LIN {X 0,Y 281.063,Z 426.792,A -85,B 0,C 180,E1 12589.746,E2 12589.746} C_VEL
LIN {X 0,Y 283.096,Z 428.214,A -85,B 0,C 180,E1 12587.55,E2 12587.55} C_VEL
LIN {X 0,Y 285.507,Z 432.072,A -85,B 0,C 180,E1 12585.18,E2 12585.18} C_VEL
LIN {X 0,Y 287.987,Z 434.4,A -85,B 0,C 180,E1 12583.244,E2 12583.244} C_VEL
LIN {X 0,Y 291.212,Z 438.721,A -85,B 0,C 180,E1 12580.955,E2 12580.955} C_VEL
LIN {X 0,Y 292.622,Z 440.371,A -85,B 0,C 180,E1 12580.065,E2 12580.065} C_VEL
LIN {X 0,Y 296.342,Z 445.028,A -85,B 0,C 180,E1 12577.894,E2 12577.894} C_VEL
LIN {X 0,Y 301.456,Z 452.142,A -85,B 0,C 180,E1 12575.238,E2 12575.238} C_VEL
LIN {X 0,Y 306.819,Z 459.539,A -85,B 0,C 180,E1 12572.796,E2 12572.796} C_VEL
LIN {X 0,Y 313.495,Z 471.371,A -85,B 0,C 180,E1 12569.997,E2 12569.997} C_VEL
LIN {X 0,Y 320.303,Z 484.326,A -85,B 0,C 180,E1 12567.438,E2 12567.438} C_VEL
LIN {X 0,Y 324.467,Z 493.018,A -85,B 0,C 180,E1 12565.976,E2 12565.976} C_VEL
LIN {X 0,Y 324.937,Z 495.745,A -85,B 0,C 180,E1 12565.75,E2 12565.75} C_VEL
LIN {X 0,Y 324.322,Z 500.372,A -85,B 0,C 180,E1 12565.731,E2 12565.731} C_VEL
LIN {X 0,Y 320.258,Z 513.224,A -85,B 0,C 180,E1 12566.295,E2 12566.295} C_VEL
LIN {X 0,Y 319.782,Z 516.489,A -85,B 0,C 180,E1 12566.293,E2 12566.293} C_VEL
LIN {X 0,Y 311.091,Z 643.63,A -85,B 0,C 180,E1 12563.53,E2 12563.53} C_VEL
LIN {X 0,Y 308.318,Z 665.175,A -85,B 0,C 180,E1 12562.857,E2 12562.857} C_VEL
LIN {X 0,Y 304.957,Z 682.984,A -85,B 0,C 180,E1 12562.072,E2 12562.072} C_VEL
LIN {X 0,Y 301.16,Z 699.447,A -85,B 0,C 180,E1 12561.128,E2 12561.128} C_VEL
LIN {X 0,Y 296.032,Z 718.293,A -85,B 0,C 180,E1 12559.756,E2 12559.756} C_VEL
LIN {X 0,Y 290.238,Z 736.04,A -85,B 0,C 180,E1 12558.081,E2 12558.081} C_VEL
LIN {X 0,Y 285.027,Z 750.363,A -85,B 0,C 180,E1 12556.437,E2 12556.437} C_VEL
LIN {X 0,Y 278.742,Z 766.216,A -85,B 0,C 180,E1 12554.239,E2 12554.239} C_VEL
LIN {X 0,Y 271.755,Z 782.159,A -85,B 0,C 180,E1 12551.472,E2 12551.472} C_VEL
LIN {X 0,Y 266.062,Z 794.478,A -85,B 0,C 180,E1 12548.871,E2 12548.871} C_VEL
LIN {X 0,Y 259.825,Z 807.626,A -85,B 0,C 180,E1 12545.525,E2 12545.525} C_VEL
LIN {X 0,Y 254.077,Z 819.333,A -85,B 0,C 180,E1 12541.775,E2 12541.775} C_VEL
LIN {X 0,Y 249.789,Z 828.338,A -85,B 0,C 180,E1 12538.27,E2 12538.27} C_VEL
LIN {X 0,Y 245.803,Z 837.325,A -85,B 0,C 180,E1 12534.002,E2 12534.002} C_VEL
LIN {X 0,Y 242.846,Z 844.673,A -85,B 0,C 180,E1 12529.445,E2 12529.445} C_VEL
LIN {X 0,Y 241.192,Z 849.808,A -85,B 0,C 180,E1 12525.385,E2 12525.385} C_VEL
LIN {X 0,Y 240.239,Z 854.173,A -85,B 0,C 180,E1 12520.788,E2 12520.788} C_VEL
LIN {X 0,Y 239.969,Z 856.979,A -85,B 0,C 180,E1 12515.979,E2 12515.979} C_VEL
LIN {X 0,Y 239.985,Z 858.077,A -85,B 0,C 180,E1 12512.149,E2 12512.149} C_VEL
LIN {X 0,Y 239.995,Z 858.167,A -85,B 0,C 180,E1 12508.568,E2 12508.568} C_VEL
LIN {X 0,Y 239.966,Z 857.285,A -85,B 0,C 180,E1 12504.836,E2 12504.836} C_VEL
LIN {X 0,Y 240.065,Z 855.439,A -85,B 0,C 180,E1 12501.136,E2 12501.136} C_VEL
LIN {X 0,Y 240.583,Z 852.272,A -85,B 0,C 180,E1 12497.031,E2 12497.031} C_VEL
LIN {X 0,Y 242.18,Z 846.644,A -85,B 0,C 180,E1 12491.963,E2 12491.963} C_VEL
LIN {X 0,Y 244.58,Z 840.152,A -85,B 0,C 180,E1 12487.655,E2 12487.655} C_VEL
LIN {X 0,Y 247.831,Z 832.624,A -85,B 0,C 180,E1 12483.655,E2 12483.655} C_VEL
LIN {X 0,Y 252.943,Z 821.703,A -85,B 0,C 180,E1 12479.079,E2 12479.079} C_VEL
LIN {X 0,Y 257.756,Z 811.744,A -85,B 0,C 180,E1 12475.726,E2 12475.726} C_VEL
LIN {X 0,Y 263.28,Z 800.376,A -85,B 0,C 180,E1 12472.545,E2 12472.545} C_VEL
LIN {X 0,Y 270.176,Z 785.665,A -85,B 0,C 180,E1 12469.219,E2 12469.219} C_VEL
LIN {X 0,Y 276.002,Z 772.517,A -85,B 0,C 180,E1 12466.791,E2 12466.791} C_VEL
LIN {X 0,Y 282.337,Z 757.376,A -85,B 0,C 180,E1 12464.474,E2 12464.474} C_VEL
LIN {X 0,Y 288.83,Z 740.076,A -85,B 0,C 180,E1 12462.348,E2 12462.348} C_VEL
LIN {X 0,Y 293.964,Z 724.757,A -85,B 0,C 180,E1 12460.82,E2 12460.82} C_VEL
LIN {X 0,Y 298.845,Z 708.319,A -85,B 0,C 180,E1 12459.479,E2 12459.479} C_VEL
LIN {X 0,Y 303.971,Z 687.7,A -85,B 0,C 180,E1 12458.175,E2 12458.175} C_VEL
LIN {X 0,Y 307.421,Z 670.269,A -85,B 0,C 180,E1 12457.351,E2 12457.351} C_VEL
LIN {X 0,Y 310.141,Z 652.377,A -85,B 0,C 180,E1 12456.715,E2 12456.715} C_VEL
LIN {X 0,Y 312.495,Z 625.497,A -85,B 0,C 180,E1 12456.047,E2 12456.047} C_VEL
LIN {X 0,Y 320.903,Z 498.988,A -85,B 0,C 180,E1 12453.315,E2 12453.315} C_VEL
LIN {X 0,Y 314.641,Z 485.874,A -85,B 0,C 180,E1 12450.991,E2 12450.991} C_VEL
LIN {X 0,Y 307.924,Z 473.075,A -85,B 0,C 180,E1 12448.253,E2 12448.253} C_VEL
LIN {X 0,Y 303.272,Z 465.071,A -85,B 0,C 180,E1 12446.172,E2 12446.172} C_VEL
LIN {X 0,Y 297.362,Z 456.629,A -85,B 0,C 180,E1 12443.279,E2 12443.279} C_VEL
LIN {X 0,Y 293.549,Z 451.571,A -85,B 0,C 180,E1 12441.172,E2 12441.172} C_VEL
LIN {X 0,Y 289.811,Z 446.551,A -85,B 0,C 180,E1 12438.827,E2 12438.827} C_VEL
LIN {X 0,Y 286.373,Z 441.99,A -85,B 0,C 180,E1 12436.331,E2 12436.331} C_VEL
LIN {X 0,Y 282.436,Z 437.446,A -85,B 0,C 180,E1 12432.895,E2 12432.895} C_VEL
LIN {X 0,Y 281.366,Z 435.538,A -85,B 0,C 180,E1 12431.695,E2 12431.695} C_VEL
LIN {X 0,Y 278.26,Z 432.838,A -85,B 0,C 180,E1 12427.649,E2 12427.649} C_VEL
LIN {X 0,Y 276.894,Z 429.844,A -85,B 0,C 180,E1 12424.358,E2 12424.358} C_VEL
LIN {X 0,Y 276.092,Z 429.238,A -85,B 0,C 180,E1 12420.009,E2 12420.009} C_VEL
LIN {X 0,Y 276.821,Z 429.756,A -85,B 0,C 180,E1 12415.452,E2 12415.452} C_VEL
LIN {X 0,Y 280.254,Z 434.876,A -85,B 0,C 180,E1 12409.11,E2 12409.11} C_VEL
LIN {X 0,Y 281.805,Z 436.112,A -85,B 0,C 180,E1 12407.406,E2 12407.406} C_VEL
LIN {X 0,Y 284.403,Z 440.099,A -85,B 0,C 180,E1 12404.826,E2 12404.826} C_VEL
LIN {X 0,Y 286.349,Z 442.006,A -85,B 0,C 180,E1 12403.268,E2 12403.268} C_VEL
LIN {X 0,Y 289.491,Z 446.297,A -85,B 0,C 180,E1 12400.961,E2 12400.961} C_VEL
LIN {X 0,Y 290.943,Z 448.031,A -85,B 0,C 180,E1 12400.015,E2 12400.015} C_VEL
LIN {X 0,Y 295.057,Z 453.594,A -85,B 0,C 180,E1 12397.549,E2 12397.549} C_VEL
LIN {X 0,Y 301.079,Z 461.013,A -85,B 0,C 180,E1 12394.487,E2 12394.487} C_VEL
LIN {X 0,Y 306.421,Z 466.113,A -85,B 0,C 180,E1 12392.197,E2 12392.197} C_VEL
LIN {X 0,Y 312.519,Z 471.944,A -85,B 0,C 180,E1 12389.647,E2 12389.647} C_VEL
LIN {X 0,Y 317.174,Z 475.591,A -85,B 0,C 180,E1 12387.606,E2 12387.606} C_VEL
LIN {X 0,Y 322.098,Z 480.221,A -85,B 0,C 180,E1 12385.18,E2 12385.18} C_VEL
LIN {X 0,Y 325.293,Z 482.787,A -85,B 0,C 180,E1 12383.517,E2 12383.517} C_VEL
LIN {X 0,Y 329.435,Z 487.109,A -85,B 0,C 180,E1 12381.091,E2 12381.091} C_VEL
LIN {X 0,Y 332.913,Z 490.098,A -85,B 0,C 180,E1 12379,E2 12379} C_VEL
LIN {X 0,Y 337.324,Z 494.746,A -85,B 0,C 180,E1 12376.216,E2 12376.216} C_VEL
LIN {X 0,Y 340.322,Z 497.124,A -85,B 0,C 180,E1 12374.339,E2 12374.339} C_VEL
LIN {X 0,Y 344.324,Z 501.472,A -85,B 0,C 180,E1 12371.633,E2 12371.633} C_VEL
LIN {X 0,Y 348.17,Z 504.479,A -85,B 0,C 180,E1 12369.047,E2 12369.047} C_VEL
LIN {X 0,Y 352.251,Z 508.897,A -85,B 0,C 180,E1 12366.023,E2 12366.023} C_VEL
LIN {X 0,Y 356.277,Z 511.889,A -85,B 0,C 180,E1 12362.972,E2 12362.972} C_VEL
LIN {X 0,Y 359.522,Z 515.605,A -85,B 0,C 180,E1 12360.223,E2 12360.223} C_VEL
LIN {X 0,Y 362.97,Z 518.189,A -85,B 0,C 180,E1 12357.21,E2 12357.21} C_VEL
LIN {X 0,Y 364.703,Z 519.278,A -85,B 0,C 180,E1 12355.606,E2 12355.606} C_VEL
LIN {X 0,Y 367.351,Z 522.689,A -85,B 0,C 180,E1 12352.705,E2 12352.705} C_VEL
LIN {X 0,Y 370.191,Z 525.054,A -85,B 0,C 180,E1 12349.403,E2 12349.403} C_VEL
LIN {X 0,Y 372.765,Z 526.313,A -85,B 0,C 180,E1 12346.037,E2 12346.037} C_VEL
LIN {X 0,Y 373.961,Z 527.419,A -85,B 0,C 180,E1 12344.081,E2 12344.081} C_VEL
LIN {X 0,Y 375.427,Z 529.663,A -85,B 0,C 180,E1 12341.055,E2 12341.055} C_VEL
LIN {X 0,Y 376.685,Z 531.057,A -85,B 0,C 180,E1 12337.78,E2 12337.78} C_VEL
LIN {X 0,Y 377.57,Z 531.82,A -85,B 0,C 180,E1 12334.404,E2 12334.404} C_VEL
LIN {X 0,Y 377.93,Z 532.086,A -85,B 0,C 180,E1 12330.975,E2 12330.975} C_VEL
LIN {X 0,Y 377.84,Z 532.043,A -85,B 0,C 180,E1 12327.573,E2 12327.573} C_VEL
LIN {X 0,Y 377.25,Z 531.557,A -85,B 0,C 180,E1 12324.22,E2 12324.22} C_VEL
LIN {X 0,Y 376.186,Z 530.598,A -85,B 0,C 180,E1 12320.824,E2 12320.824} C_VEL
LIN {X 0,Y 374.776,Z 528.735,A -85,B 0,C 180,E1 12317.49,E2 12317.49} C_VEL
LIN {X 0,Y 373.168,Z 526.505,A -85,B 0,C 180,E1 12314.618,E2 12314.618} C_VEL
LIN {X 0,Y 370.673,Z 525.343,A -85,B 0,C 180,E1 12311.192,E2 12311.192} C_VEL
LIN {X 0,Y 367.915,Z 523.228,A -85,B 0,C 180,E1 12307.9,E2 12307.9} C_VEL
LIN {X 0,Y 365.196,Z 520.086,A -85,B 0,C 180,E1 12304.965,E2 12304.965} C_VEL
LIN {X 0,Y 364.121,Z 518.785,A -85,B 0,C 180,E1 12303.863,E2 12303.863} C_VEL
LIN {X 0,Y 360.72,Z 516.653,A -85,B 0,C 180,E1 12300.802,E2 12300.802} C_VEL
LIN {X 0,Y 357.303,Z 513.23,A -85,B 0,C 180,E1 12297.882,E2 12297.882} C_VEL
LIN {X 0,Y 355.438,Z 511.103,A -85,B 0,C 180,E1 12296.354,E2 12296.354} C_VEL
LIN {X 0,Y 351.656,Z 508.36,A -85,B 0,C 180,E1 12293.542,E2 12293.542} C_VEL
LIN {X 0,Y 347.13,Z 503.534,A -85,B 0,C 180,E1 12290.251,E2 12290.251} C_VEL
LIN {X 0,Y 342.897,Z 500.119,A -85,B 0,C 180,E1 12287.399,E2 12287.399} C_VEL
LIN {X 0,Y 339.244,Z 496.148,A -85,B 0,C 180,E1 12284.982,E2 12284.982} C_VEL
LIN {X 0,Y 335.113,Z 492.634,A -85,B 0,C 180,E1 12282.386,E2 12282.386} C_VEL
LIN {X 0,Y 331.562,Z 488.792,A -85,B 0,C 180,E1 12280.178,E2 12280.178} C_VEL
LIN {X 0,Y 326.988,Z 484.774,A -85,B 0,C 180,E1 12277.468,E2 12277.468} C_VEL
LIN {X 0,Y 324.177,Z 481.699,A -85,B 0,C 180,E1 12275.862,E2 12275.862} C_VEL
LIN {X 0,Y 319.289,Z 477.796,A -85,B 0,C 180,E1 12273.434,E2 12273.434} C_VEL
LIN {X 0,Y 315.454,Z 474.122,A -85,B 0,C 180,E1 12271.627,E2 12271.627} C_VEL
LIN {X 0,Y 310.125,Z 469.815,A -85,B 0,C 180,E1 12269.333,E2 12269.333} C_VEL
LIN {X 0,Y 305.78,Z 465.642,A -85,B 0,C 180,E1 12267.549,E2 12267.549} C_VEL
LIN {X 0,Y 300.52,Z 460.302,A -85,B 0,C 180,E1 12265.247,E2 12265.247} C_VEL
LIN {X 0,Y 297.512,Z 456.84,A -85,B 0,C 180,E1 12263.773,E2 12263.773} C_VEL
LIN {X 0,Y 293.368,Z 451.342,A -85,B 0,C 180,E1 12261.482,E2 12261.482} C_VEL
LIN {X 0,Y 289.931,Z 446.705,A -85,B 0,C 180,E1 12259.323,E2 12259.323} C_VEL
LIN {X 0,Y 286.583,Z 442.444,A -85,B 0,C 180,E1 12256.927,E2 12256.927} C_VEL
LIN {X 0,Y 285.74,Z 441.229,A -85,B 0,C 180,E1 12256.246,E2 12256.246} C_VEL
LIN {X 0,Y 282.707,Z 437.891,A -85,B 0,C 180,E1 12253.593,E2 12253.593} C_VEL
LIN {X 0,Y 281.539,Z 435.676,A -85,B 0,C 180,E1 12252.293,E2 12252.293} C_VEL
LIN {X 0,Y 278.028,Z 432.465,A -85,B 0,C 180,E1 12247.637,E2 12247.637} C_VEL
LIN {X 0,Y 276.821,Z 429.756,A -85,B 0,C 180,E1 12244.548,E2 12244.548} C_VEL
LIN {X 0,Y 276.119,Z 429.246,A -85,B 0,C 180,E1 12239.369,E2 12239.369} C_VEL
LIN {X 0,Y 276.962,Z 429.954,A -85,B 0,C 180,E1 12235.436,E2 12235.436} C_VEL
LIN {X 0,Y 279.77,Z 434.54,A -85,B 0,C 180,E1 12230.114,E2 12230.114} C_VEL
LIN {X 0,Y 281.732,Z 435.981,A -85,B 0,C 180,E1 12227.905,E2 12227.905} C_VEL
LIN {X 0,Y 284.193,Z 439.881,A -85,B 0,C 180,E1 12225.423,E2 12225.423} C_VEL
LIN {X 0,Y 286.432,Z 442.099,A -85,B 0,C 180,E1 12223.62,E2 12223.62} C_VEL
LIN {X 0,Y 289.811,Z 446.551,A -85,B 0,C 180,E1 12221.173,E2 12221.173} C_VEL
LIN {X 0,Y 295.249,Z 453.802,A -85,B 0,C 180,E1 12217.86,E2 12217.86} C_VEL
LIN {X 0,Y 299.195,Z 459.285,A -85,B 0,C 180,E1 12215.775,E2 12215.775} C_VEL
LIN {X 0,Y 304.238,Z 466.464,A -85,B 0,C 180,E1 12213.392,E2 12213.392} C_VEL
LIN {X 0,Y 310.55,Z 477.957,A -85,B 0,C 180,E1 12210.64,E2 12210.64} C_VEL
LIN {X 0,Y 317.191,Z 490.983,A -85,B 0,C 180,E1 12208.043,E2 12208.043} C_VEL
LIN {X 0,Y 320.95,Z 499.412,A -85,B 0,C 180,E1 12206.656,E2 12206.656} C_VEL
LIN {X 0,Y 319.782,Z 516.489,A -85,B 0,C 180,E1 12206.293,E2 12206.293} C_VEL
LIN {X 0,Y 318.718,Z 524.178,A -85,B 0,C 180,E1 12206.273,E2 12206.273} C_VEL
LIN {X 0,Y 313.81,Z 544.667,A -85,B 0,C 180,E1 12206.786,E2 12206.786} C_VEL
LIN {X 0,Y 312.937,Z 551.268,A -85,B 0,C 180,E1 12206.759,E2 12206.759} C_VEL
LIN {X 0,Y 306.362,Z 643.68,A -85,B 0,C 180,E1 12204.729,E2 12204.729} C_VEL
LIN {X 0,Y 303.411,Z 665.624,A -85,B 0,C 180,E1 12204.038,E2 12204.038} C_VEL
LIN {X 0,Y 299.976,Z 683.221,A -85,B 0,C 180,E1 12203.259,E2 12203.259} C_VEL
LIN {X 0,Y 296.024,Z 699.782,A -85,B 0,C 180,E1 12202.305,E2 12202.305} C_VEL
LIN {X 0,Y 290.568,Z 718.989,A -85,B 0,C 180,E1 12200.89,E2 12200.89} C_VEL
LIN {X 0,Y 284.887,Z 735.801,A -85,B 0,C 180,E1 12199.294,E2 12199.294} C_VEL
LIN {X 0,Y 279.449,Z 750.226,A -85,B 0,C 180,E1 12197.632,E2 12197.632} C_VEL
LIN {X 0,Y 272.706,Z 766.606,A -85,B 0,C 180,E1 12195.338,E2 12195.338} C_VEL
LIN {X 0,Y 265.686,Z 781.918,A -85,B 0,C 180,E1 12192.639,E2 12192.639} C_VEL
LIN {X 0,Y 259.655,Z 794.397,A -85,B 0,C 180,E1 12189.968,E2 12189.968} C_VEL
LIN {X 0,Y 253.19,Z 807.383,A -85,B 0,C 180,E1 12186.604,E2 12186.604} C_VEL
LIN {X 0,Y 247.185,Z 818.975,A -85,B 0,C 180,E1 12182.821,E2 12182.821} C_VEL
LIN {X 0,Y 242.758,Z 827.729,A -85,B 0,C 180,E1 12179.348,E2 12179.348} C_VEL
LIN {X 0,Y 238.524,Z 836.624,A -85,B 0,C 180,E1 12175.047,E2 12175.047} C_VEL
LIN {X 0,Y 235.296,Z 844.047,A -85,B 0,C 180,E1 12170.392,E2 12170.392} C_VEL
LIN {X 0,Y 233.422,Z 849.294,A -85,B 0,C 180,E1 12166.166,E2 12166.166} C_VEL
LIN {X 0,Y 232.39,Z 853.297,A -85,B 0,C 180,E1 12161.918,E2 12161.918} C_VEL
LIN {X 0,Y 231.98,Z 856.561,A -85,B 0,C 180,E1 12156.683,E2 12156.683} C_VEL
LIN {X 0,Y 231.983,Z 857.81,A -85,B 0,C 180,E1 12152.47,E2 12152.47} C_VEL
LIN {X 0,Y 232.001,Z 857.96,A -85,B 0,C 180,E1 12148.765,E2 12148.765} C_VEL
LIN {X 0,Y 231.968,Z 857.102,A -85,B 0,C 180,E1 12144.807,E2 12144.807} C_VEL
LIN {X 0,Y 232.087,Z 855.2,A -85,B 0,C 180,E1 12140.828,E2 12140.828} C_VEL
LIN {X 0,Y 232.668,Z 852.032,A -85,B 0,C 180,E1 12136.582,E2 12136.582} C_VEL
LIN {X 0,Y 234.469,Z 846.245,A -85,B 0,C 180,E1 12131.227,E2 12131.227} C_VEL
LIN {X 0,Y 237.019,Z 839.889,A -85,B 0,C 180,E1 12126.889,E2 12126.889} C_VEL
LIN {X 0,Y 240.495,Z 832.381,A -85,B 0,C 180,E1 12122.786,E2 12122.786} C_VEL
LIN {X 0,Y 245.928,Z 821.461,A -85,B 0,C 180,E1 12118.095,E2 12118.095} C_VEL
LIN {X 0,Y 250.946,Z 811.627,A -85,B 0,C 180,E1 12114.71,E2 12114.71} C_VEL
LIN {X 0,Y 256.763,Z 800.245,A -85,B 0,C 180,E1 12111.462,E2 12111.462} C_VEL
LIN {X 0,Y 264.073,Z 785.34,A -85,B 0,C 180,E1 12108.043,E2 12108.043} C_VEL
LIN {X 0,Y 270.124,Z 772.25,A -85,B 0,C 180,E1 12105.602,E2 12105.602} C_VEL
LIN {X 0,Y 276.699,Z 757.135,A -85,B 0,C 180,E1 12103.272,E2 12103.272} C_VEL
LIN {X 0,Y 283.49,Z 739.677,A -85,B 0,C 180,E1 12101.12,E2 12101.12} C_VEL
LIN {X 0,Y 288.743,Z 724.517,A -85,B 0,C 180,E1 12099.606,E2 12099.606} C_VEL
LIN {X 0,Y 293.609,Z 708.663,A -85,B 0,C 180,E1 12098.308,E2 12098.308} C_VEL
LIN {X 0,Y 298.854,Z 688.443,A -85,B 0,C 180,E1 12097.015,E2 12097.015} C_VEL
LIN {X 0,Y 302.585,Z 670.198,A -85,B 0,C 180,E1 12096.149,E2 12096.149} C_VEL
LIN {X 0,Y 305.37,Z 652.435,A -85,B 0,C 180,E1 12095.518,E2 12095.518} C_VEL
LIN {X 0,Y 307.827,Z 625.458,A -85,B 0,C 180,E1 12094.844,E2 12094.844} C_VEL
LIN {X 0,Y 316.271,Z 502.394,A -85,B 0,C 180,E1 12092.168,E2 12092.168} C_VEL
LIN {X 0,Y 309.873,Z 488.932,A -85,B 0,C 180,E1 12089.643,E2 12089.643} C_VEL
LIN {X 0,Y 304.035,Z 477.659,A -85,B 0,C 180,E1 12087.103,E2 12087.103} C_VEL
LIN {X 0,Y 300.474,Z 471.542,A -85,B 0,C 180,E1 12085.428,E2 12085.428} C_VEL
LIN {X 0,Y 294.834,Z 463.361,A -85,B 0,C 180,E1 12082.54,E2 12082.54} C_VEL
LIN {X 0,Y 291.623,Z 458.938,A -85,B 0,C 180,E1 12080.687,E2 12080.687} C_VEL
LIN {X 0,Y 287.983,Z 453.959,A -85,B 0,C 180,E1 12078.321,E2 12078.321} C_VEL
LIN {X 0,Y 284.164,Z 448.891,A -85,B 0,C 180,E1 12075.406,E2 12075.406} C_VEL
LIN {X 0,Y 280.975,Z 444.988,A -85,B 0,C 180,E1 12072.441,E2 12072.441} C_VEL
LIN {X 0,Y 280.213,Z 443.419,A -85,B 0,C 180,E1 12071.535,E2 12071.535} C_VEL
LIN {X 0,Y 277.055,Z 440.544,A -85,B 0,C 180,E1 12067.265,E2 12067.265} C_VEL
LIN {X 0,Y 275.787,Z 437.642,A -85,B 0,C 180,E1 12063.959,E2 12063.959} C_VEL
LIN {X 0,Y 275.202,Z 437.187,A -85,B 0,C 180,E1 12058.344,E2 12058.344} C_VEL
LIN {X 0,Y 275.975,Z 437.963,A -85,B 0,C 180,E1 12055.021,E2 12055.021} C_VEL
LIN {X 0,Y 278.479,Z 442.248,A -85,B 0,C 180,E1 12050.086,E2 12050.086} C_VEL
LIN {X 0,Y 280.454,Z 443.854,A -85,B 0,C 180,E1 12047.763,E2 12047.763} C_VEL
LIN {X 0,Y 283.093,Z 447.906,A -85,B 0,C 180,E1 12045.069,E2 12045.069} C_VEL
LIN {X 0,Y 284.81,Z 449.701,A -85,B 0,C 180,E1 12043.647,E2 12043.647} C_VEL
LIN {X 0,Y 288.101,Z 454.126,A -85,B 0,C 180,E1 12041.181,E2 12041.181} C_VEL
LIN {X 0,Y 293.014,Z 460.861,A -85,B 0,C 180,E1 12038.07,E2 12038.07} C_VEL
LIN {X 0,Y 302.783,Z 472.331,A -85,B 0,C 180,E1 12033.219,E2 12033.219} C_VEL
LIN {X 0,Y 306.521,Z 475.768,A -85,B 0,C 180,E1 12031.677,E2 12031.677} C_VEL
LIN {X 0,Y 312.244,Z 480.744,A -85,B 0,C 180,E1 12029.298,E2 12029.298} C_VEL
LIN {X 0,Y 315.511,Z 483.383,A -85,B 0,C 180,E1 12027.845,E2 12027.845} C_VEL
LIN {X 0,Y 320.718,Z 488.088,A -85,B 0,C 180,E1 12025.335,E2 12025.335} C_VEL
LIN {X 0,Y 323.777,Z 490.587,A -85,B 0,C 180,E1 12023.758,E2 12023.758} C_VEL
LIN {X 0,Y 328.075,Z 494.935,A -85,B 0,C 180,E1 12021.277,E2 12021.277} C_VEL
LIN {X 0,Y 331.331,Z 497.7,A -85,B 0,C 180,E1 12019.334,E2 12019.334} C_VEL
LIN {X 0,Y 335.745,Z 502.367,A -85,B 0,C 180,E1 12016.548,E2 12016.548} C_VEL
LIN {X 0,Y 338.95,Z 504.965,A -85,B 0,C 180,E1 12014.544,E2 12014.544} C_VEL
LIN {X 0,Y 343.103,Z 509.355,A -85,B 0,C 180,E1 12011.768,E2 12011.768} C_VEL
LIN {X 0,Y 346.764,Z 512.216,A -85,B 0,C 180,E1 12009.298,E2 12009.298} C_VEL
LIN {X 0,Y 350.89,Z 516.636,A -85,B 0,C 180,E1 12006.271,E2 12006.271} C_VEL
LIN {X 0,Y 355.015,Z 519.713,A -85,B 0,C 180,E1 12003.171,E2 12003.171} C_VEL
LIN {X 0,Y 358.273,Z 523.392,A -85,B 0,C 180,E1 12000.44,E2 12000.44} C_VEL
LIN {X 0,Y 361.677,Z 525.992,A -85,B 0,C 180,E1 11997.474,E2 11997.474} C_VEL
LIN {X 0,Y 363.669,Z 527.353,A -85,B 0,C 180,E1 11995.63,E2 11995.63} C_VEL
LIN {X 0,Y 366.427,Z 530.758,A -85,B 0,C 180,E1 11992.627,E2 11992.627} C_VEL
LIN {X 0,Y 369.294,Z 533.068,A -85,B 0,C 180,E1 11989.287,E2 11989.287} C_VEL
LIN {X 0,Y 371.857,Z 534.284,A -85,B 0,C 180,E1 11985.917,E2 11985.917} C_VEL
LIN {X 0,Y 373.032,Z 535.52,A -85,B 0,C 180,E1 11983.959,E2 11983.959} C_VEL
LIN {X 0,Y 374.509,Z 537.68,A -85,B 0,C 180,E1 11980.926,E2 11980.926} C_VEL
LIN {X 0,Y 375.738,Z 539.057,A -85,B 0,C 180,E1 11977.646,E2 11977.646} C_VEL
LIN {X 0,Y 376.594,Z 539.761,A -85,B 0,C 180,E1 11974.416,E2 11974.416} C_VEL
LIN {X 0,Y 376.95,Z 540.022,A -85,B 0,C 180,E1 11971.064,E2 11971.064} C_VEL
LIN {X 0,Y 376.881,Z 540.001,A -85,B 0,C 180,E1 11967.719,E2 11967.719} C_VEL
LIN {X 0,Y 376.303,Z 539.536,A -85,B 0,C 180,E1 11964.358,E2 11964.358} C_VEL
LIN {X 0,Y 375.259,Z 538.596,A -85,B 0,C 180,E1 11960.956,E2 11960.956} C_VEL
LIN {X 0,Y 373.858,Z 536.835,A -85,B 0,C 180,E1 11957.646,E2 11957.646} C_VEL
LIN {X 0,Y 372.159,Z 534.437,A -85,B 0,C 180,E1 11954.575,E2 11954.575} C_VEL
LIN {X 0,Y 369.666,Z 533.282,A -85,B 0,C 180,E1 11951.17,E2 11951.17} C_VEL
LIN {X 0,Y 366.905,Z 531.193,A -85,B 0,C 180,E1 11947.873,E2 11947.873} C_VEL
LIN {X 0,Y 364.168,Z 528.127,A -85,B 0,C 180,E1 11944.939,E2 11944.939} C_VEL
LIN {X 0,Y 362.912,Z 526.633,A -85,B 0,C 180,E1 11943.669,E2 11943.669} C_VEL
LIN {X 0,Y 359.595,Z 524.555,A -85,B 0,C 180,E1 11940.702,E2 11940.702} C_VEL
LIN {X 0,Y 356.059,Z 521.038,A -85,B 0,C 180,E1 11937.679,E2 11937.679} C_VEL
LIN {X 0,Y 354.264,Z 518.975,A -85,B 0,C 180,E1 11936.221,E2 11936.221} C_VEL
LIN {X 0,Y 350.444,Z 516.229,A -85,B 0,C 180,E1 11933.396,E2 11933.396} C_VEL
LIN {X 0,Y 345.757,Z 511.302,A -85,B 0,C 180,E1 11930.009,E2 11930.009} C_VEL
LIN {X 0,Y 341.499,Z 507.866,A -85,B 0,C 180,E1 11927.159,E2 11927.159} C_VEL
LIN {X 0,Y 337.844,Z 503.908,A -85,B 0,C 180,E1 11924.744,E2 11924.744} C_VEL
LIN {X 0,Y 333.528,Z 500.234,A -85,B 0,C 180,E1 11922.054,E2 11922.054} C_VEL
LIN {X 0,Y 330.109,Z 496.537,A -85,B 0,C 180,E1 11919.937,E2 11919.937} C_VEL
LIN {X 0,Y 325.364,Z 492.372,A -85,B 0,C 180,E1 11917.134,E2 11917.134} C_VEL
LIN {X 0,Y 322.273,Z 489.205,A -85,B 0,C 180,E1 11915.45,E2 11915.45} C_VEL
LIN {X 0,Y 317.515,Z 485.391,A -85,B 0,C 180,E1 11913.111,E2 11913.111} C_VEL
LIN {X 0,Y 313.418,Z 481.576,A -85,B 0,C 180,E1 11911.213,E2 11911.213} C_VEL
LIN {X 0,Y 307.553,Z 476.797,A -85,B 0,C 180,E1 11908.749,E2 11908.749} C_VEL
LIN {X 0,Y 303.4,Z 472.851,A -85,B 0,C 180,E1 11907.039,E2 11907.039} C_VEL
LIN {X 0,Y 298.11,Z 467.242,A -85,B 0,C 180,E1 11904.636,E2 11904.636} C_VEL
LIN {X 0,Y 292.359,Z 459.775,A -85,B 0,C 180,E1 11901.533,E2 11901.533} C_VEL
LIN {X 0,Y 288.101,Z 454.126,A -85,B 0,C 180,E1 11898.819,E2 11898.819} C_VEL
LIN {X 0,Y 284.754,Z 449.593,A -85,B 0,C 180,E1 11896.304,E2 11896.304} C_VEL
LIN {X 0,Y 280.956,Z 444.916,A -85,B 0,C 180,E1 11892.831,E2 11892.831} C_VEL
LIN {X 0,Y 280.193,Z 443.453,A -85,B 0,C 180,E1 11891.935,E2 11891.935} C_VEL
LIN {X 0,Y 276.739,Z 439.992,A -85,B 0,C 180,E1 11887.047,E2 11887.047} C_VEL
LIN {X 0,Y 275.781,Z 437.647,A -85,B 0,C 180,E1 11884.357,E2 11884.357} C_VEL
LIN {X 0,Y 275.177,Z 437.212,A -85,B 0,C 180,E1 11878.95,E2 11878.95} C_VEL
LIN {X 0,Y 275.983,Z 437.959,A -85,B 0,C 180,E1 11875.42,E2 11875.42} C_VEL
LIN {X 0,Y 278.488,Z 442.289,A -85,B 0,C 180,E1 11870.485,E2 11870.485} C_VEL
LIN {X 0,Y 280.381,Z 443.728,A -85,B 0,C 180,E1 11868.264,E2 11868.264} C_VEL
LIN {X 0,Y 282.997,Z 447.807,A -85,B 0,C 180,E1 11865.569,E2 11865.569} C_VEL
LIN {X 0,Y 284.891,Z 449.782,A -85,B 0,C 180,E1 11864,E2 11864} C_VEL
LIN {X 0,Y 289.102,Z 455.481,A -85,B 0,C 180,E1 11860.916,E2 11860.916} C_VEL
LIN {X 0,Y 293.358,Z 461.31,A -85,B 0,C 180,E1 11858.289,E2 11858.289} C_VEL
LIN {X 0,Y 297.31,Z 466.941,A -85,B 0,C 180,E1 11856.139,E2 11856.139} C_VEL
LIN {X 0,Y 301.782,Z 473.558,A -85,B 0,C 180,E1 11853.953,E2 11853.953} C_VEL
LIN {X 0,Y 307.646,Z 484.541,A -85,B 0,C 180,E1 11851.295,E2 11851.295} C_VEL
LIN {X 0,Y 314.228,Z 497.864,A -85,B 0,C 180,E1 11848.618,E2 11848.618} C_VEL
LIN {X 0,Y 316.343,Z 502.92,A -85,B 0,C 180,E1 11847.79,E2 11847.79} C_VEL
LIN {X 0,Y 312.937,Z 551.268,A -85,B 0,C 180,E1 11846.759,E2 11846.759} C_VEL
LIN {X 0,Y 311.858,Z 558.957,A -85,B 0,C 180,E1 11846.744,E2 11846.744} C_VEL
LIN {X 0,Y 306.979,Z 579.443,A -85,B 0,C 180,E1 11847.274,E2 11847.274} C_VEL
LIN {X 0,Y 306.093,Z 586.044,A -85,B 0,C 180,E1 11847.251,E2 11847.251} C_VEL
LIN {X 0,Y 301.715,Z 644.337,A -85,B 0,C 180,E1 11845.951,E2 11845.951} C_VEL
LIN {X 0,Y 298.51,Z 666.76,A -85,B 0,C 180,E1 11845.229,E2 11845.229} C_VEL
LIN {X 0,Y 294.952,Z 684.249,A -85,B 0,C 180,E1 11844.445,E2 11844.445} C_VEL
LIN {X 0,Y 290.341,Z 702.727,A -85,B 0,C 180,E1 11843.357,E2 11843.357} C_VEL
LIN {X 0,Y 284.592,Z 721.515,A -85,B 0,C 180,E1 11841.902,E2 11841.902} C_VEL
LIN {X 0,Y 279.066,Z 737.175,A -85,B 0,C 180,E1 11840.38,E2 11840.38} C_VEL
LIN {X 0,Y 272.896,Z 752.834,A -85,B 0,C 180,E1 11838.525,E2 11838.525} C_VEL
LIN {X 0,Y 265.145,Z 770.349,A -85,B 0,C 180,E1 11835.919,E2 11835.919} C_VEL
LIN {X 0,Y 258.987,Z 783.179,A -85,B 0,C 180,E1 11833.559,E2 11833.559} C_VEL
LIN {X 0,Y 252.611,Z 795.779,A -85,B 0,C 180,E1 11830.773,E2 11830.773} C_VEL
LIN {X 0,Y 245.195,Z 809.731,A -85,B 0,C 180,E1 11826.93,E2 11826.93} C_VEL
LIN {X 0,Y 239.683,Z 819.905,A -85,B 0,C 180,E1 11823.443,E2 11823.443} C_VEL
LIN {X 0,Y 234.522,Z 829.663,A -85,B 0,C 180,E1 11819.359,E2 11819.359} C_VEL
LIN {X 0,Y 230.062,Z 838.46,A -85,B 0,C 180,E1 11814.658,E2 11814.658} C_VEL
LIN {X 0,Y 227.202,Z 844.815,A -85,B 0,C 180,E1 11810.344,E2 11810.344} C_VEL
LIN {X 0,Y 225.25,Z 850.144,A -85,B 0,C 180,E1 11805.71,E2 11805.71} C_VEL
LIN {X 0,Y 224.181,Z 854.511,A -85,B 0,C 180,E1 11800.276,E2 11800.276} C_VEL
LIN {X 0,Y 223.971,Z 856.684,A -85,B 0,C 180,E1 11795.893,E2 11795.893} C_VEL
LIN {X 0,Y 223.993,Z 857.634,A -85,B 0,C 180,E1 11792.046,E2 11792.046} C_VEL
LIN {X 0,Y 224,Z 857.694,A -85,B 0,C 180,E1 11788.465,E2 11788.465} C_VEL
LIN {X 0,Y 223.97,Z 856.864,A -85,B 0,C 180,E1 11784.621,E2 11784.621} C_VEL
LIN {X 0,Y 224.111,Z 854.962,A -85,B 0,C 180,E1 11780.499,E2 11780.499} C_VEL
LIN {X 0,Y 224.763,Z 851.791,A -85,B 0,C 180,E1 11776.101,E2 11776.101} C_VEL
LIN {X 0,Y 226.678,Z 846.161,A -85,B 0,C 180,E1 11770.682,E2 11770.682} C_VEL
LIN {X 0,Y 229.481,Z 839.667,A -85,B 0,C 180,E1 11766.097,E2 11766.097} C_VEL
LIN {X 0,Y 233.217,Z 832.139,A -85,B 0,C 180,E1 11761.863,E2 11761.863} C_VEL
LIN {X 0,Y 238.989,Z 821.218,A -85,B 0,C 180,E1 11757.053,E2 11757.053} C_VEL
LIN {X 0,Y 244.288,Z 811.385,A -85,B 0,C 180,E1 11753.597,E2 11753.597} C_VEL
LIN {X 0,Y 250.404,Z 800.002,A -85,B 0,C 180,E1 11750.293,E2 11750.293} C_VEL
LIN {X 0,Y 258.008,Z 785.182,A -85,B 0,C 180,E1 11746.845,E2 11746.845} C_VEL
LIN {X 0,Y 264.346,Z 772.035,A -85,B 0,C 180,E1 11744.369,E2 11744.369} C_VEL
LIN {X 0,Y 271.19,Z 756.895,A -85,B 0,C 180,E1 11742.021,E2 11742.021} C_VEL
LIN {X 0,Y 278.167,Z 739.596,A -85,B 0,C 180,E1 11739.88,E2 11739.88} C_VEL
LIN {X 0,Y 283.61,Z 724.415,A -85,B 0,C 180,E1 11738.359,E2 11738.359} C_VEL
LIN {X 0,Y 288.689,Z 708.387,A -85,B 0,C 180,E1 11737.049,E2 11737.049} C_VEL
LIN {X 0,Y 294.115,Z 688.043,A -85,B 0,C 180,E1 11735.754,E2 11735.754} C_VEL
LIN {X 0,Y 297.894,Z 670.085,A -85,B 0,C 180,E1 11734.906,E2 11734.906} C_VEL
LIN {X 0,Y 300.757,Z 652.345,A -85,B 0,C 180,E1 11734.278,E2 11734.278} C_VEL
LIN {X 0,Y 303.299,Z 625.418,A -85,B 0,C 180,E1 11733.604,E2 11733.604} C_VEL
LIN {X 0,Y 311.81,Z 506.063,A -85,B 0,C 180,E1 11731.011,E2 11731.011} C_VEL
LIN {X 0,Y 305.373,Z 492.254,A -85,B 0,C 180,E1 11728.298,E2 11728.298} C_VEL
LIN {X 0,Y 299.806,Z 481.496,A -85,B 0,C 180,E1 11725.7,E2 11725.7} C_VEL
LIN {X 0,Y 296.052,Z 475.426,A -85,B 0,C 180,E1 11723.81,E2 11723.81} C_VEL
LIN {X 0,Y 290.34,Z 467.002,A -85,B 0,C 180,E1 11720.572,E2 11720.572} C_VEL
LIN {X 0,Y 286.041,Z 461.213,A -85,B 0,C 180,E1 11717.712,E2 11717.712} C_VEL
LIN {X 0,Y 282.609,Z 456.496,A -85,B 0,C 180,E1 11714.976,E2 11714.976} C_VEL
LIN {X 0,Y 279.533,Z 452.53,A -85,B 0,C 180,E1 11711.982,E2 11711.982} C_VEL
LIN {X 0,Y 278.691,Z 451.108,A -85,B 0,C 180,E1 11710.97,E2 11710.97} C_VEL
LIN {X 0,Y 275.764,Z 448.066,A -85,B 0,C 180,E1 11706.671,E2 11706.671} C_VEL
LIN {X 0,Y 274.749,Z 445.535,A -85,B 0,C 180,E1 11703.765,E2 11703.765} C_VEL
LIN {X 0,Y 274.314,Z 445.176,A -85,B 0,C 180,E1 11697.711,E2 11697.711} C_VEL
LIN {X 0,Y 274.987,Z 446.038,A -85,B 0,C 180,E1 11695.003,E2 11695.003} C_VEL
LIN {X 0,Y 277.359,Z 450.127,A -85,B 0,C 180,E1 11690.255,E2 11690.255} C_VEL
LIN {X 0,Y 279.115,Z 451.589,A -85,B 0,C 180,E1 11688.123,E2 11688.123} C_VEL
LIN {X 0,Y 281.789,Z 455.711,A -85,B 0,C 180,E1 11685.314,E2 11685.314} C_VEL
LIN {X 0,Y 283.286,Z 457.383,A -85,B 0,C 180,E1 11684.03,E2 11684.03} C_VEL
LIN {X 0,Y 286.715,Z 461.951,A -85,B 0,C 180,E1 11681.403,E2 11681.403} C_VEL
LIN {X 0,Y 291.304,Z 468.614,A -85,B 0,C 180,E1 11678.411,E2 11678.411} C_VEL
LIN {X 0,Y 297.281,Z 476.211,A -85,B 0,C 180,E1 11675.203,E2 11675.203} C_VEL
LIN {X 0,Y 308.692,Z 487.066,A -85,B 0,C 180,E1 11670.304,E2 11670.304} C_VEL
LIN {X 0,Y 313.461,Z 490.779,A -85,B 0,C 180,E1 11668.256,E2 11668.256} C_VEL
LIN {X 0,Y 318.633,Z 495.412,A -85,B 0,C 180,E1 11665.839,E2 11665.839} C_VEL
LIN {X 0,Y 322.097,Z 498.193,A -85,B 0,C 180,E1 11664.09,E2 11664.09} C_VEL
LIN {X 0,Y 326.413,Z 502.502,A -85,B 0,C 180,E1 11661.642,E2 11661.642} C_VEL
LIN {X 0,Y 329.985,Z 505.613,A -85,B 0,C 180,E1 11659.509,E2 11659.509} C_VEL
LIN {X 0,Y 334.624,Z 510.36,A -85,B 0,C 180,E1 11656.602,E2 11656.602} C_VEL
LIN {X 0,Y 337.533,Z 512.741,A -85,B 0,C 180,E1 11654.782,E2 11654.782} C_VEL
LIN {X 0,Y 341.869,Z 517.224,A -85,B 0,C 180,E1 11651.914,E2 11651.914} C_VEL
LIN {X 0,Y 345.537,Z 520.165,A -85,B 0,C 180,E1 11649.428,E2 11649.428} C_VEL
LIN {X 0,Y 349.823,Z 524.628,A -85,B 0,C 180,E1 11646.31,E2 11646.31} C_VEL
LIN {X 0,Y 353.744,Z 527.528,A -85,B 0,C 180,E1 11643.376,E2 11643.376} C_VEL
LIN {X 0,Y 357.047,Z 531.198,A -85,B 0,C 180,E1 11640.64,E2 11640.64} C_VEL
LIN {X 0,Y 360.543,Z 533.881,A -85,B 0,C 180,E1 11637.588,E2 11637.588} C_VEL
LIN {X 0,Y 362.435,Z 535.148,A -85,B 0,C 180,E1 11635.84,E2 11635.84} C_VEL
LIN {X 0,Y 365.201,Z 538.529,A -85,B 0,C 180,E1 11632.877,E2 11632.877} C_VEL
LIN {X 0,Y 368.132,Z 540.907,A -85,B 0,C 180,E1 11629.515,E2 11629.515} C_VEL
LIN {X 0,Y 370.735,Z 542.174,A -85,B 0,C 180,E1 11626.128,E2 11626.128} C_VEL
LIN {X 0,Y 371.874,Z 543.209,A -85,B 0,C 180,E1 11624.321,E2 11624.321} C_VEL
LIN {X 0,Y 373.36,Z 545.468,A -85,B 0,C 180,E1 11621.273,E2 11621.273} C_VEL
LIN {X 0,Y 374.687,Z 546.885,A -85,B 0,C 180,E1 11617.976,E2 11617.976} C_VEL
LIN {X 0,Y 375.578,Z 547.677,A -85,B 0,C 180,E1 11614.581,E2 11614.581} C_VEL
LIN {X 0,Y 375.967,Z 547.973,A -85,B 0,C 180,E1 11611.219,E2 11611.219} C_VEL
LIN {X 0,Y 375.944,Z 547.974,A -85,B 0,C 180,E1 11608.019,E2 11608.019} C_VEL
LIN {X 0,Y 375.39,Z 547.546,A -85,B 0,C 180,E1 11604.651,E2 11604.651} C_VEL
LIN {X 0,Y 374.335,Z 546.588,A -85,B 0,C 180,E1 11601.088,E2 11601.088} C_VEL
LIN {X 0,Y 372.929,Z 544.902,A -85,B 0,C 180,E1 11597.772,E2 11597.772} C_VEL
LIN {X 0,Y 371.15,Z 542.368,A -85,B 0,C 180,E1 11594.532,E2 11594.532} C_VEL
LIN {X 0,Y 368.66,Z 541.221,A -85,B 0,C 180,E1 11591.147,E2 11591.147} C_VEL
LIN {X 0,Y 365.888,Z 539.154,A -85,B 0,C 180,E1 11587.846,E2 11587.846} C_VEL
LIN {X 0,Y 363.056,Z 536.038,A -85,B 0,C 180,E1 11584.819,E2 11584.819} C_VEL
LIN {X 0,Y 361.78,Z 534.517,A -85,B 0,C 180,E1 11583.542,E2 11583.542} C_VEL
LIN {X 0,Y 358.35,Z 532.361,A -85,B 0,C 180,E1 11580.499,E2 11580.499} C_VEL
LIN {X 0,Y 354.713,Z 528.757,A -85,B 0,C 180,E1 11577.419,E2 11577.419} C_VEL
LIN {X 0,Y 353.055,Z 526.826,A -85,B 0,C 180,E1 11576.058,E2 11576.058} C_VEL
LIN {X 0,Y 349.099,Z 523.976,A -85,B 0,C 180,E1 11573.153,E2 11573.153} C_VEL
LIN {X 0,Y 344.389,Z 519.068,A -85,B 0,C 180,E1 11569.763,E2 11569.763} C_VEL
LIN {X 0,Y 339.95,Z 515.466,A -85,B 0,C 180,E1 11566.822,E2 11566.822} C_VEL
LIN {X 0,Y 336.428,Z 511.661,A -85,B 0,C 180,E1 11564.5,E2 11564.5} C_VEL
LIN {X 0,Y 331.934,Z 507.834,A -85,B 0,C 180,E1 11561.722,E2 11561.722} C_VEL
LIN {X 0,Y 328.616,Z 504.251,A -85,B 0,C 180,E1 11559.667,E2 11559.667} C_VEL
LIN {X 0,Y 323.902,Z 500.181,A -85,B 0,C 180,E1 11556.919,E2 11556.919} C_VEL
LIN {X 0,Y 320.536,Z 496.819,A -85,B 0,C 180,E1 11555.123,E2 11555.123} C_VEL
LIN {X 0,Y 315.37,Z 492.623,A -85,B 0,C 180,E1 11552.602,E2 11552.602} C_VEL
LIN {X 0,Y 311.358,Z 489.019,A -85,B 0,C 180,E1 11550.799,E2 11550.799} C_VEL
LIN {X 0,Y 305.383,Z 484.166,A -85,B 0,C 180,E1 11548.331,E2 11548.331} C_VEL
LIN {X 0,Y 301.045,Z 480.053,A -85,B 0,C 180,E1 11546.522,E2 11546.522} C_VEL
LIN {X 0,Y 295.675,Z 474.094,A -85,B 0,C 180,E1 11543.983,E2 11543.983} C_VEL
LIN {X 0,Y 290.395,Z 467.117,A -85,B 0,C 180,E1 11541.024,E2 11541.024} C_VEL
LIN {X 0,Y 286.293,Z 461.539,A -85,B 0,C 180,E1 11538.309,E2 11538.309} C_VEL
LIN {X 0,Y 282.597,Z 456.448,A -85,B 0,C 180,E1 11535.378,E2 11535.378} C_VEL
LIN {X 0,Y 279.61,Z 452.647,A -85,B 0,C 180,E1 11532.484,E2 11532.484} C_VEL
LIN {X 0,Y 278.859,Z 451.224,A -85,B 0,C 180,E1 11531.573,E2 11531.573} C_VEL
LIN {X 0,Y 275.568,Z 447.698,A -85,B 0,C 180,E1 11526.658,E2 11526.658} C_VEL
LIN {X 0,Y 274.743,Z 445.541,A -85,B 0,C 180,E1 11524.165,E2 11524.165} C_VEL
LIN {X 0,Y 274.252,Z 445.17,A -85,B 0,C 180,E1 11518.529,E2 11518.529} C_VEL
LIN {X 0,Y 274.936,Z 445.842,A -85,B 0,C 180,E1 11515.611,E2 11515.611} C_VEL
LIN {X 0,Y 277.218,Z 450.036,A -85,B 0,C 180,E1 11510.86,E2 11510.86} C_VEL
LIN {X 0,Y 279.121,Z 451.65,A -85,B 0,C 180,E1 11508.524,E2 11508.524} C_VEL
LIN {X 0,Y 281.804,Z 455.729,A -85,B 0,C 180,E1 11505.716,E2 11505.716} C_VEL
LIN {X 0,Y 283.363,Z 457.455,A -85,B 0,C 180,E1 11504.384,E2 11504.384} C_VEL
LIN {X 0,Y 287.402,Z 463.08,A -85,B 0,C 180,E1 11501.325,E2 11501.325} C_VEL
LIN {X 0,Y 291.563,Z 468.927,A -85,B 0,C 180,E1 11498.677,E2 11498.677} C_VEL
LIN {X 0,Y 296.76,Z 476.421,A -85,B 0,C 180,E1 11495.828,E2 11495.828} C_VEL
LIN {X 0,Y 300.355,Z 482.489,A -85,B 0,C 180,E1 11494.032,E2 11494.032} C_VEL
LIN {X 0,Y 305.663,Z 492.885,A -85,B 0,C 180,E1 11491.572,E2 11491.572} C_VEL
LIN {X 0,Y 311.868,Z 506.194,A -85,B 0,C 180,E1 11488.966,E2 11488.966} C_VEL
LIN {X 0,Y 306.093,Z 586.044,A -85,B 0,C 180,E1 11487.251,E2 11487.251} C_VEL
LIN {X 0,Y 305,Z 593.732,A -85,B 0,C 180,E1 11487.242,E2 11487.242} C_VEL
LIN {X 0,Y 300.143,Z 614.212,A -85,B 0,C 180,E1 11487.793,E2 11487.793} C_VEL
LIN {X 0,Y 299.251,Z 620.811,A -85,B 0,C 180,E1 11487.773,E2 11487.773} C_VEL
LIN {X 0,Y 296.7,Z 649.453,A -85,B 0,C 180,E1 11487.088,E2 11487.088} C_VEL
LIN {X 0,Y 293.569,Z 668.811,A -85,B 0,C 180,E1 11486.422,E2 11486.422} C_VEL
LIN {X 0,Y 290.008,Z 685.499,A -85,B 0,C 180,E1 11485.659,E2 11485.659} C_VEL
LIN {X 0,Y 284.94,Z 704.853,A -85,B 0,C 180,E1 11484.495,E2 11484.495} C_VEL
LIN {X 0,Y 279.031,Z 723.119,A -85,B 0,C 180,E1 11483.04,E2 11483.04} C_VEL
LIN {X 0,Y 273.607,Z 737.878,A -85,B 0,C 180,E1 11481.585,E2 11481.585} C_VEL
LIN {X 0,Y 266.703,Z 754.725,A -85,B 0,C 180,E1 11479.554,E2 11479.554} C_VEL
LIN {X 0,Y 259.264,Z 770.67,A -85,B 0,C 180,E1 11477.115,E2 11477.115} C_VEL
LIN {X 0,Y 252.871,Z 783.438,A -85,B 0,C 180,E1 11474.732,E2 11474.732} C_VEL
LIN {X 0,Y 245.537,Z 797.322,A -85,B 0,C 180,E1 11471.585,E2 11471.585} C_VEL
LIN {X 0,Y 238.356,Z 810.053,A -85,B 0,C 180,E1 11467.931,E2 11467.931} C_VEL
LIN {X 0,Y 232.829,Z 819.732,A -85,B 0,C 180,E1 11464.53,E2 11464.53} C_VEL
LIN {X 0,Y 227.392,Z 829.42,A -85,B 0,C 180,E1 11460.374,E2 11460.374} C_VEL
LIN {X 0,Y 222.512,Z 838.432,A -85,B 0,C 180,E1 11455.401,E2 11455.401} C_VEL
LIN {X 0,Y 219.54,Z 844.573,A -85,B 0,C 180,E1 11451.087,E2 11451.087} C_VEL
LIN {X 0,Y 217.41,Z 849.903,A -85,B 0,C 180,E1 11446.292,E2 11446.292} C_VEL
LIN {X 0,Y 216.216,Z 854.271,A -85,B 0,C 180,E1 11440.659,E2 11440.659} C_VEL
LIN {X 0,Y 215.977,Z 856.356,A -85,B 0,C 180,E1 11436.379,E2 11436.379} C_VEL
LIN {X 0,Y 215.99,Z 857.367,A -85,B 0,C 180,E1 11432.388,E2 11432.388} C_VEL
LIN {X 0,Y 216.006,Z 857.487,A -85,B 0,C 180,E1 11428.674,E2 11428.674} C_VEL
LIN {X 0,Y 215.972,Z 856.627,A -85,B 0,C 180,E1 11424.421,E2 11424.421} C_VEL
LIN {X 0,Y 216.138,Z 854.723,A -85,B 0,C 180,E1 11420.145,E2 11420.145} C_VEL
LIN {X 0,Y 216.888,Z 851.5,A -85,B 0,C 180,E1 11415.52,E2 11415.52} C_VEL
LIN {X 0,Y 219.107,Z 845.582,A -85,B 0,C 180,E1 11409.708,E2 11409.708} C_VEL
LIN {X 0,Y 222,Z 839.425,A -85,B 0,C 180,E1 11405.238,E2 11405.238} C_VEL
LIN {X 0,Y 226.002,Z 831.896,A -85,B 0,C 180,E1 11400.88,E2 11400.88} C_VEL
LIN {X 0,Y 232.134,Z 820.975,A -85,B 0,C 180,E1 11395.949,E2 11395.949} C_VEL
LIN {X 0,Y 237.729,Z 811.142,A -85,B 0,C 180,E1 11392.423,E2 11392.423} C_VEL
LIN {X 0,Y 244.156,Z 799.76,A -85,B 0,C 180,E1 11389.065,E2 11389.065} C_VEL
LIN {X 0,Y 252.176,Z 784.8,A -85,B 0,C 180,E1 11385.546,E2 11385.546} C_VEL
LIN {X 0,Y 258.712,Z 771.794,A -85,B 0,C 180,E1 11383.079,E2 11383.079} C_VEL
LIN {X 0,Y 265.813,Z 756.659,A -85,B 0,C 180,E1 11380.72,E2 11380.72} C_VEL
LIN {X 0,Y 273.042,Z 739.357,A -85,B 0,C 180,E1 11378.575,E2 11378.575} C_VEL
LIN {X 0,Y 278.678,Z 724.133,A -85,B 0,C 180,E1 11377.051,E2 11377.051} C_VEL
LIN {X 0,Y 283.937,Z 708.043,A -85,B 0,C 180,E1 11375.741,E2 11375.741} C_VEL
LIN {X 0,Y 289.67,Z 686.987,A -85,B 0,C 180,E1 11374.418,E2 11374.418} C_VEL
LIN {X 0,Y 293.457,Z 669.401,A -85,B 0,C 180,E1 11373.602,E2 11373.602} C_VEL
LIN {X 0,Y 296.441,Z 651.223,A -85,B 0,C 180,E1 11372.968,E2 11372.968} C_VEL
LIN {X 0,Y 299.01,Z 624.109,A -85,B 0,C 180,E1 11372.299,E2 11372.299} C_VEL
LIN {X 0,Y 307.428,Z 509.52,A -85,B 0,C 180,E1 11369.795,E2 11369.795} C_VEL
LIN {X 0,Y 301.303,Z 496.355,A -85,B 0,C 180,E1 11367.048,E2 11367.048} C_VEL
LIN {X 0,Y 296.091,Z 486.11,A -85,B 0,C 180,E1 11364.443,E2 11364.443} C_VEL
LIN {X 0,Y 290.485,Z 477.546,A -85,B 0,C 180,E1 11361.353,E2 11361.353} C_VEL
LIN {X 0,Y 287.39,Z 473.117,A -85,B 0,C 180,E1 11359.413,E2 11359.413} C_VEL
LIN {X 0,Y 284.398,Z 468.758,A -85,B 0,C 180,E1 11357.29,E2 11357.29} C_VEL
LIN {X 0,Y 281.062,Z 464.086,A -85,B 0,C 180,E1 11354.533,E2 11354.533} C_VEL
LIN {X 0,Y 278.027,Z 459.902,A -85,B 0,C 180,E1 11351.416,E2 11351.416} C_VEL
LIN {X 0,Y 277.372,Z 458.886,A -85,B 0,C 180,E1 11350.602,E2 11350.602} C_VEL
LIN {X 0,Y 274.542,Z 455.675,A -85,B 0,C 180,E1 11346.168,E2 11346.168} C_VEL
LIN {X 0,Y 273.714,Z 453.43,A -85,B 0,C 180,E1 11343.569,E2 11343.569} C_VEL
LIN {X 0,Y 273.416,Z 453.152,A -85,B 0,C 180,E1 11337.284,E2 11337.284} C_VEL
LIN {X 0,Y 273.939,Z 453.935,A -85,B 0,C 180,E1 11335.194,E2 11335.194} C_VEL
LIN {X 0,Y 276.241,Z 458.006,A -85,B 0,C 180,E1 11330.426,E2 11330.426} C_VEL
LIN {X 0,Y 277.864,Z 459.498,A -85,B 0,C 180,E1 11328.385,E2 11328.385} C_VEL
LIN {X 0,Y 280.6,Z 463.627,A -85,B 0,C 180,E1 11325.461,E2 11325.461} C_VEL
LIN {X 0,Y 281.83,Z 465.158,A -85,B 0,C 180,E1 11324.368,E2 11324.368} C_VEL
LIN {X 0,Y 285.774,Z 470.719,A -85,B 0,C 180,E1 11321.286,E2 11321.286} C_VEL
LIN {X 0,Y 289.476,Z 476.143,A -85,B 0,C 180,E1 11318.838,E2 11318.838} C_VEL
LIN {X 0,Y 298.915,Z 487.423,A -85,B 0,C 180,E1 11313.916,E2 11313.916} C_VEL
LIN {X 0,Y 307.588,Z 495.262,A -85,B 0,C 180,E1 11310.294,E2 11310.294} C_VEL
LIN {X 0,Y 311.683,Z 498.443,A -85,B 0,C 180,E1 11308.552,E2 11308.552} C_VEL
LIN {X 0,Y 316.64,Z 502.859,A -85,B 0,C 180,E1 11306.249,E2 11306.249} C_VEL
LIN {X 0,Y 320.52,Z 505.981,A -85,B 0,C 180,E1 11304.326,E2 11304.326} C_VEL
LIN {X 0,Y 325.043,Z 510.335,A -85,B 0,C 180,E1 11301.821,E2 11301.821} C_VEL
LIN {X 0,Y 328.415,Z 513.266,A -85,B 0,C 180,E1 11299.815,E2 11299.815} C_VEL
LIN {X 0,Y 333.204,Z 518.106,A -85,B 0,C 180,E1 11296.844,E2 11296.844} C_VEL
LIN {X 0,Y 336.123,Z 520.514,A -85,B 0,C 180,E1 11295.022,E2 11295.022} C_VEL
LIN {X 0,Y 340.481,Z 524.97,A -85,B 0,C 180,E1 11292.157,E2 11292.157} C_VEL
LIN {X 0,Y 344.156,Z 527.916,A -85,B 0,C 180,E1 11289.672,E2 11289.672} C_VEL
LIN {X 0,Y 348.466,Z 532.369,A -85,B 0,C 180,E1 11286.561,E2 11286.561} C_VEL
LIN {X 0,Y 352.472,Z 535.339,A -85,B 0,C 180,E1 11283.583,E2 11283.583} C_VEL
LIN {X 0,Y 355.911,Z 539.107,A -85,B 0,C 180,E1 11280.744,E2 11280.744} C_VEL
LIN {X 0,Y 359.437,Z 541.783,A -85,B 0,C 180,E1 11277.68,E2 11277.68} C_VEL
LIN {X 0,Y 361.237,Z 542.987,A -85,B 0,C 180,E1 11276.021,E2 11276.021} C_VEL
LIN {X 0,Y 364.143,Z 546.462,A -85,B 0,C 180,E1 11272.948,E2 11272.948} C_VEL
LIN {X 0,Y 367.101,Z 548.832,A -85,B 0,C 180,E1 11269.573,E2 11269.573} C_VEL
LIN {X 0,Y 369.717,Z 550.104,A -85,B 0,C 180,E1 11266.173,E2 11266.173} C_VEL
LIN {X 0,Y 370.859,Z 551.171,A -85,B 0,C 180,E1 11264.361,E2 11264.361} C_VEL
LIN {X 0,Y 372.364,Z 553.41,A -85,B 0,C 180,E1 11261.304,E2 11261.304} C_VEL
LIN {X 0,Y 373.655,Z 554.767,A -85,B 0,C 180,E1 11258.153,E2 11258.153} C_VEL
LIN {X 0,Y 374.513,Z 555.567,A -85,B 0,C 180,E1 11254.901,E2 11254.901} C_VEL
LIN {X 0,Y 374.986,Z 555.929,A -85,B 0,C 180,E1 11251.528,E2 11251.528} C_VEL
LIN {X 0,Y 374.99,Z 555.927,A -85,B 0,C 180,E1 11248.166,E2 11248.166} C_VEL
LIN {X 0,Y 374.436,Z 555.511,A -85,B 0,C 180,E1 11244.768,E2 11244.768} C_VEL
LIN {X 0,Y 373.467,Z 554.616,A -85,B 0,C 180,E1 11241.378,E2 11241.378} C_VEL
LIN {X 0,Y 372.076,Z 553.059,A -85,B 0,C 180,E1 11238.059,E2 11238.059} C_VEL
LIN {X 0,Y 370.245,Z 550.363,A -85,B 0,C 180,E1 11234.654,E2 11234.654} C_VEL
LIN {X 0,Y 367.796,Z 549.223,A -85,B 0,C 180,E1 11231.29,E2 11231.29} C_VEL
LIN {X 0,Y 365.142,Z 547.358,A -85,B 0,C 180,E1 11228.137,E2 11228.137} C_VEL
LIN {X 0,Y 362.235,Z 544.341,A -85,B 0,C 180,E1 11225.02,E2 11225.02} C_VEL
LIN {X 0,Y 360.529,Z 542.34,A -85,B 0,C 180,E1 11223.304,E2 11223.304} C_VEL
LIN {X 0,Y 357.026,Z 540.099,A -85,B 0,C 180,E1 11220.224,E2 11220.224} C_VEL
LIN {X 0,Y 353.37,Z 536.478,A -85,B 0,C 180,E1 11217.159,E2 11217.159} C_VEL
LIN {X 0,Y 351.596,Z 534.554,A -85,B 0,C 180,E1 11215.733,E2 11215.733} C_VEL
LIN {X 0,Y 347.623,Z 531.587,A -85,B 0,C 180,E1 11212.801,E2 11212.801} C_VEL
LIN {X 0,Y 343.021,Z 526.833,A -85,B 0,C 180,E1 11209.517,E2 11209.517} C_VEL
LIN {X 0,Y 338.556,Z 523.214,A -85,B 0,C 180,E1 11206.58,E2 11206.58} C_VEL
LIN {X 0,Y 335.014,Z 519.412,A -85,B 0,C 180,E1 11204.253,E2 11204.253} C_VEL
LIN {X 0,Y 330.499,Z 515.59,A -85,B 0,C 180,E1 11201.48,E2 11201.48} C_VEL
LIN {X 0,Y 326.911,Z 511.805,A -85,B 0,C 180,E1 11199.267,E2 11199.267} C_VEL
LIN {X 0,Y 321.993,Z 507.55,A -85,B 0,C 180,E1 11196.464,E2 11196.464} C_VEL
LIN {X 0,Y 318.635,Z 504.309,A -85,B 0,C 180,E1 11194.703,E2 11194.703} C_VEL
LIN {X 0,Y 313.121,Z 499.849,A -85,B 0,C 180,E1 11192.106,E2 11192.106} C_VEL
LIN {X 0,Y 309.635,Z 496.724,A -85,B 0,C 180,E1 11190.558,E2 11190.558} C_VEL
LIN {X 0,Y 303.834,Z 492.12,A -85,B 0,C 180,E1 11188.168,E2 11188.168} C_VEL
LIN {X 0,Y 298.519,Z 487.07,A -85,B 0,C 180,E1 11185.907,E2 11185.907} C_VEL
LIN {X 0,Y 293.224,Z 480.861,A -85,B 0,C 180,E1 11183.289,E2 11183.289} C_VEL
LIN {X 0,Y 288.492,Z 474.518,A -85,B 0,C 180,E1 11180.532,E2 11180.532} C_VEL
LIN {X 0,Y 284.509,Z 468.946,A -85,B 0,C 180,E1 11177.793,E2 11177.793} C_VEL
LIN {X 0,Y 281.051,Z 464.051,A -85,B 0,C 180,E1 11174.937,E2 11174.937} C_VEL
LIN {X 0,Y 278.101,Z 460.022,A -85,B 0,C 180,E1 11171.921,E2 11171.921} C_VEL
LIN {X 0,Y 277.361,Z 458.877,A -85,B 0,C 180,E1 11171.005,E2 11171.005} C_VEL
LIN {X 0,Y 274.33,Z 455.207,A -85,B 0,C 180,E1 11166.058,E2 11166.058} C_VEL
LIN {X 0,Y 273.709,Z 453.435,A -85,B 0,C 180,E1 11163.971,E2 11163.971} C_VEL
LIN {X 0,Y 273.342,Z 453.125,A -85,B 0,C 180,E1 11158.104,E2 11158.104} C_VEL
LIN {X 0,Y 273.917,Z 453.842,A -85,B 0,C 180,E1 11155.7,E2 11155.7} C_VEL
LIN {X 0,Y 276.247,Z 458.044,A -85,B 0,C 180,E1 11150.828,E2 11150.828} C_VEL
LIN {X 0,Y 277.792,Z 459.377,A -85,B 0,C 180,E1 11148.889,E2 11148.889} C_VEL
LIN {X 0,Y 280.612,Z 463.647,A -85,B 0,C 180,E1 11145.865,E2 11145.865} C_VEL
LIN {X 0,Y 281.96,Z 465.318,A -85,B 0,C 180,E1 11144.674,E2 11144.674} C_VEL
LIN {X 0,Y 285.651,Z 470.56,A -85,B 0,C 180,E1 11141.788,E2 11141.788} C_VEL
LIN {X 0,Y 289.629,Z 476.301,A -85,B 0,C 180,E1 11139.164,E2 11139.164} C_VEL
LIN {X 0,Y 294.61,Z 483.738,A -85,B 0,C 180,E1 11136.332,E2 11136.332} C_VEL
LIN {X 0,Y 298.027,Z 489.705,A -85,B 0,C 180,E1 11134.561,E2 11134.561} C_VEL
LIN {X 0,Y 303.677,Z 501.326,A -85,B 0,C 180,E1 11131.851,E2 11131.851} C_VEL
LIN {X 0,Y 307.508,Z 510.015,A -85,B 0,C 180,E1 11130.157,E2 11130.157} C_VEL
LIN {X 0,Y 299.251,Z 620.811,A -85,B 0,C 180,E1 11127.773,E2 11127.773} C_VEL
LIN {X 0,Y 298.137,Z 628.498,A -85,B 0,C 180,E1 11127.773,E2 11127.773} C_VEL
LIN {X 0,Y 293.094,Z 647.805,A -85,B 0,C 180,E1 11128.304,E2 11128.304} C_VEL
LIN {X 0,Y 291.489,Z 655.403,A -85,B 0,C 180,E1 11128.214,E2 11128.214} C_VEL
LIN {X 0,Y 288.072,Z 674.411,A -85,B 0,C 180,E1 11127.512,E2 11127.512} C_VEL
LIN {X 0,Y 283.097,Z 694.782,A -85,B 0,C 180,E1 11126.459,E2 11126.459} C_VEL
LIN {X 0,Y 278.276,Z 710.994,A -85,B 0,C 180,E1 11125.364,E2 11125.364} C_VEL
LIN {X 0,Y 272.6,Z 727.487,A -85,B 0,C 180,E1 11123.973,E2 11123.973} C_VEL
LIN {X 0,Y 264.946,Z 746.529,A -85,B 0,C 180,E1 11121.921,E2 11121.921} C_VEL
LIN {X 0,Y 258.47,Z 760.834,A -85,B 0,C 180,E1 11119.988,E2 11119.988} C_VEL
LIN {X 0,Y 251.24,Z 775.485,A -85,B 0,C 180,E1 11117.579,E2 11117.579} C_VEL
LIN {X 0,Y 242.956,Z 790.833,A -85,B 0,C 180,E1 11114.394,E2 11114.394} C_VEL
LIN {X 0,Y 236.143,Z 802.694,A -85,B 0,C 180,E1 11111.338,E2 11111.338} C_VEL
LIN {X 0,Y 228.821,Z 815.119,A -85,B 0,C 180,E1 11107.399,E2 11107.399} C_VEL
LIN {X 0,Y 222.242,Z 825.912,A -85,B 0,C 180,E1 11102.981,E2 11102.981} C_VEL
LIN {X 0,Y 217.475,Z 834.01,A -85,B 0,C 180,E1 11098.864,E2 11098.864} C_VEL
LIN {X 0,Y 212.964,Z 842.311,A -85,B 0,C 180,E1 11093.519,E2 11093.519} C_VEL
LIN {X 0,Y 210.123,Z 848.297,A -85,B 0,C 180,E1 11088.303,E2 11088.303} C_VEL
LIN {X 0,Y 208.665,Z 852.366,A -85,B 0,C 180,E1 11083.579,E2 11083.579} C_VEL
LIN {X 0,Y 208.025,Z 855.666,A -85,B 0,C 180,E1 11078.002,E2 11078.002} C_VEL
LIN {X 0,Y 207.989,Z 857.1,A -85,B 0,C 180,E1 11072.755,E2 11072.755} C_VEL
LIN {X 0,Y 208.008,Z 857.251,A -85,B 0,C 180,E1 11068.623,E2 11068.623} C_VEL
LIN {X 0,Y 207.973,Z 856.47,A -85,B 0,C 180,E1 11064.453,E2 11064.453} C_VEL
LIN {X 0,Y 208.147,Z 854.624,A -85,B 0,C 180,E1 11060.023,E2 11060.023} C_VEL
LIN {X 0,Y 208.924,Z 851.522,A -85,B 0,C 180,E1 11055.307,E2 11055.307} C_VEL
LIN {X 0,Y 211.011,Z 846.349,A -85,B 0,C 180,E1 11049.764,E2 11049.764} C_VEL
LIN {X 0,Y 214.356,Z 839.584,A -85,B 0,C 180,E1 11044.588,E2 11044.588} C_VEL
LIN {X 0,Y 218.291,Z 832.596,A -85,B 0,C 180,E1 11040.352,E2 11040.352} C_VEL
LIN {X 0,Y 224.156,Z 822.847,A -85,B 0,C 180,E1 11035.623,E2 11035.623} C_VEL
LIN {X 0,Y 230.857,Z 811.604,A -85,B 0,C 180,E1 11031.416,E2 11031.416} C_VEL
LIN {X 0,Y 237.076,Z 801.106,A -85,B 0,C 180,E1 11028.215,E2 11028.215} C_VEL
LIN {X 0,Y 245.025,Z 787.202,A -85,B 0,C 180,E1 11024.764,E2 11024.764} C_VEL
LIN {X 0,Y 252.645,Z 772.676,A -85,B 0,C 180,E1 11021.927,E2 11021.927} C_VEL
LIN {X 0,Y 259.371,Z 758.94,A -85,B 0,C 180,E1 11019.733,E2 11019.733} C_VEL
LIN {X 0,Y 267.112,Z 741.539,A -85,B 0,C 180,E1 11017.483,E2 11017.483} C_VEL
LIN {X 0,Y 273.585,Z 724.723,A -85,B 0,C 180,E1 11015.776,E2 11015.776} C_VEL
LIN {X 0,Y 278.69,Z 709.703,A -85,B 0,C 180,E1 11014.539,E2 11014.539} C_VEL
LIN {X 0,Y 283.804,Z 692.293,A -85,B 0,C 180,E1 11013.39,E2 11013.39} C_VEL
LIN {X 0,Y 288.626,Z 671.549,A -85,B 0,C 180,E1 11012.372,E2 11012.372} C_VEL
LIN {X 0,Y 291.687,Z 654.083,A -85,B 0,C 180,E1 11011.745,E2 11011.745} C_VEL
LIN {X 0,Y 294.051,Z 633.688,A -85,B 0,C 180,E1 11011.195,E2 11011.195} C_VEL
LIN {X 0,Y 303.224,Z 513.265,A -85,B 0,C 180,E1 11008.57,E2 11008.57} C_VEL
LIN {X 0,Y 296.941,Z 499.509,A -85,B 0,C 180,E1 11005.538,E2 11005.538} C_VEL
LIN {X 0,Y 292.987,Z 491.895,A -85,B 0,C 180,E1 11003.434,E2 11003.434} C_VEL
LIN {X 0,Y 288.016,Z 484.132,A -85,B 0,C 180,E1 11000.533,E2 11000.533} C_VEL
LIN {X 0,Y 285.26,Z 480.098,A -85,B 0,C 180,E1 10998.714,E2 10998.714} C_VEL
LIN {X 0,Y 282.641,Z 476.151,A -85,B 0,C 180,E1 10996.765,E2 10996.765} C_VEL
LIN {X 0,Y 279.533,Z 471.671,A -85,B 0,C 180,E1 10994.085,E2 10994.085} C_VEL
LIN {X 0,Y 276.625,Z 467.445,A -85,B 0,C 180,E1 10990.947,E2 10990.947} C_VEL
LIN {X 0,Y 275.899,Z 466.545,A -85,B 0,C 180,E1 10990.026,E2 10990.026} C_VEL
LIN {X 0,Y 273.271,Z 463.111,A -85,B 0,C 180,E1 10985.468,E2 10985.468} C_VEL
LIN {X 0,Y 272.682,Z 461.327,A -85,B 0,C 180,E1 10983.372,E2 10983.372} C_VEL
LIN {X 0,Y 272.484,Z 461.12,A -85,B 0,C 180,E1 10977.065,E2 10977.065} C_VEL
LIN {X 0,Y 272.921,Z 461.937,A -85,B 0,C 180,E1 10975.281,E2 10975.281} C_VEL
LIN {X 0,Y 275.126,Z 465.884,A -85,B 0,C 180,E1 10970.598,E2 10970.598} C_VEL
LIN {X 0,Y 276.545,Z 467.221,A -85,B 0,C 180,E1 10968.751,E2 10968.751} C_VEL
LIN {X 0,Y 279.304,Z 471.431,A -85,B 0,C 180,E1 10965.71,E2 10965.71} C_VEL
LIN {X 0,Y 280.386,Z 472.919,A -85,B 0,C 180,E1 10964.71,E2 10964.71} C_VEL
LIN {X 0,Y 284.041,Z 478.196,A -85,B 0,C 180,E1 10961.753,E2 10961.753} C_VEL
LIN {X 0,Y 287.622,Z 483.604,A -85,B 0,C 180,E1 10959.296,E2 10959.296} C_VEL
LIN {X 0,Y 296.802,Z 494.794,A -85,B 0,C 180,E1 10954.36,E2 10954.36} C_VEL
LIN {X 0,Y 305.886,Z 502.978,A -85,B 0,C 180,E1 10950.543,E2 10950.543} C_VEL
LIN {X 0,Y 310.139,Z 506.335,A -85,B 0,C 180,E1 10948.744,E2 10948.744} C_VEL
LIN {X 0,Y 315.392,Z 510.865,A -85,B 0,C 180,E1 10946.316,E2 10946.316} C_VEL
LIN {X 0,Y 318.838,Z 513.652,A -85,B 0,C 180,E1 10944.619,E2 10944.619} C_VEL
LIN {X 0,Y 323.231,Z 517.811,A -85,B 0,C 180,E1 10942.244,E2 10942.244} C_VEL
LIN {X 0,Y 326.866,Z 520.934,A -85,B 0,C 180,E1 10940.115,E2 10940.115} C_VEL
LIN {X 0,Y 331.641,Z 525.729,A -85,B 0,C 180,E1 10937.182,E2 10937.182} C_VEL
LIN {X 0,Y 334.802,Z 528.397,A -85,B 0,C 180,E1 10935.202,E2 10935.202} C_VEL
LIN {X 0,Y 339.227,Z 532.84,A -85,B 0,C 180,E1 10932.3,E2 10932.3} C_VEL
LIN {X 0,Y 342.781,Z 535.667,A -85,B 0,C 180,E1 10929.918,E2 10929.918} C_VEL
LIN {X 0,Y 347.117,Z 540.116,A -85,B 0,C 180,E1 10926.807,E2 10926.807} C_VEL
LIN {X 0,Y 351.209,Z 543.155,A -85,B 0,C 180,E1 10923.787,E2 10923.787} C_VEL
LIN {X 0,Y 354.569,Z 546.837,A -85,B 0,C 180,E1 10921.011,E2 10921.011} C_VEL
LIN {X 0,Y 358.101,Z 549.556,A -85,B 0,C 180,E1 10917.973,E2 10917.973} C_VEL
LIN {X 0,Y 360.042,Z 550.825,A -85,B 0,C 180,E1 10916.202,E2 10916.202} C_VEL
LIN {X 0,Y 363.005,Z 554.317,A -85,B 0,C 180,E1 10913.106,E2 10913.106} C_VEL
LIN {X 0,Y 365.918,Z 556.664,A -85,B 0,C 180,E1 10909.805,E2 10909.805} C_VEL
LIN {X 0,Y 368.57,Z 557.991,A -85,B 0,C 180,E1 10906.387,E2 10906.387} C_VEL
LIN {X 0,Y 369.736,Z 558.989,A -85,B 0,C 180,E1 10904.566,E2 10904.566} C_VEL
LIN {X 0,Y 371.305,Z 561.28,A -85,B 0,C 180,E1 10901.478,E2 10901.478} C_VEL
LIN {X 0,Y 372.604,Z 562.649,A -85,B 0,C 180,E1 10898.332,E2 10898.332} C_VEL
LIN {X 0,Y 373.496,Z 563.481,A -85,B 0,C 180,E1 10895.068,E2 10895.068} C_VEL
LIN {X 0,Y 374.012,Z 563.872,A -85,B 0,C 180,E1 10891.685,E2 10891.685} C_VEL
LIN {X 0,Y 374.013,Z 563.873,A -85,B 0,C 180,E1 10888.315,E2 10888.315} C_VEL
LIN {X 0,Y 373.495,Z 563.481,A -85,B 0,C 180,E1 10884.932,E2 10884.932} C_VEL
LIN {X 0,Y 372.605,Z 562.648,A -85,B 0,C 180,E1 10881.668,E2 10881.668} C_VEL
LIN {X 0,Y 371.298,Z 561.273,A -85,B 0,C 180,E1 10878.506,E2 10878.506} C_VEL
LIN {X 0,Y 369.633,Z 558.844,A -85,B 0,C 180,E1 10875.27,E2 10875.27} C_VEL
LIN {X 0,Y 368.36,Z 557.918,A -85,B 0,C 180,E1 10873.331,E2 10873.331} C_VEL
LIN {X 0,Y 365.633,Z 556.468,A -85,B 0,C 180,E1 10869.846,E2 10869.846} C_VEL
LIN {X 0,Y 362.735,Z 554.04,A -85,B 0,C 180,E1 10866.593,E2 10866.593} C_VEL
LIN {X 0,Y 359.851,Z 550.549,A -85,B 0,C 180,E1 10863.605,E2 10863.605} C_VEL
LIN {X 0,Y 356.226,Z 548.26,A -85,B 0,C 180,E1 10860.397,E2 10860.397} C_VEL
LIN {X 0,Y 352.52,Z 544.77,A -85,B 0,C 180,E1 10857.296,E2 10857.296} C_VEL
LIN {X 0,Y 350.336,Z 542.385,A -85,B 0,C 180,E1 10855.55,E2 10855.55} C_VEL
LIN {X 0,Y 346.451,Z 539.51,A -85,B 0,C 180,E1 10852.696,E2 10852.696} C_VEL
LIN {X 0,Y 341.581,Z 534.572,A -85,B 0,C 180,E1 10849.252,E2 10849.252} C_VEL
LIN {X 0,Y 337.066,Z 530.873,A -85,B 0,C 180,E1 10846.28,E2 10846.28} C_VEL
LIN {X 0,Y 333.305,Z 526.987,A -85,B 0,C 180,E1 10843.851,E2 10843.851} C_VEL
LIN {X 0,Y 328.76,Z 523.022,A -85,B 0,C 180,E1 10841.043,E2 10841.043} C_VEL
LIN {X 0,Y 325.375,Z 519.488,A -85,B 0,C 180,E1 10838.974,E2 10838.974} C_VEL
LIN {X 0,Y 320.499,Z 515.325,A -85,B 0,C 180,E1 10836.228,E2 10836.228} C_VEL
LIN {X 0,Y 316.898,Z 511.918,A -85,B 0,C 180,E1 10834.374,E2 10834.374} C_VEL
LIN {X 0,Y 311.451,Z 507.603,A -85,B 0,C 180,E1 10831.865,E2 10831.865} C_VEL
LIN {X 0,Y 307.357,Z 504.052,A -85,B 0,C 180,E1 10830.084,E2 10830.084} C_VEL
LIN {X 0,Y 301.013,Z 498.893,A -85,B 0,C 180,E1 10827.486,E2 10827.486} C_VEL
LIN {X 0,Y 292.058,Z 489.466,A -85,B 0,C 180,E1 10823.281,E2 10823.281} C_VEL
LIN {X 0,Y 284.77,Z 479.356,A -85,B 0,C 180,E1 10818.782,E2 10818.782} C_VEL
LIN {X 0,Y 282.75,Z 476.347,A -85,B 0,C 180,E1 10817.269,E2 10817.269} C_VEL
LIN {X 0,Y 279.523,Z 471.645,A -85,B 0,C 180,E1 10814.49,E2 10814.49} C_VEL
LIN {X 0,Y 276.697,Z 467.567,A -85,B 0,C 180,E1 10811.454,E2 10811.454} C_VEL
LIN {X 0,Y 276.057,Z 466.636,A -85,B 0,C 180,E1 10810.635,E2 10810.635} C_VEL
LIN {X 0,Y 273.158,Z 462.808,A -85,B 0,C 180,E1 10805.557,E2 10805.557} C_VEL
LIN {X 0,Y 272.678,Z 461.33,A -85,B 0,C 180,E1 10803.775,E2 10803.775} C_VEL
LIN {X 0,Y 272.445,Z 461.092,A -85,B 0,C 180,E1 10797.677,E2 10797.677} C_VEL
LIN {X 0,Y 272.894,Z 461.877,A -85,B 0,C 180,E1 10795.789,E2 10795.789} C_VEL
LIN {X 0,Y 275.13,Z 465.922,A -85,B 0,C 180,E1 10791.001,E2 10791.001} C_VEL
LIN {X 0,Y 276.55,Z 467.272,A -85,B 0,C 180,E1 10789.155,E2 10789.155} C_VEL
LIN {X 0,Y 279.423,Z 471.561,A -85,B 0,C 180,E1 10786.015,E2 10786.015} C_VEL
LIN {X 0,Y 280.731,Z 473.446,A -85,B 0,C 180,E1 10784.816,E2 10784.816} C_VEL
LIN {X 0,Y 283.92,Z 478.036,A -85,B 0,C 180,E1 10782.257,E2 10782.257} C_VEL
LIN {X 0,Y 287.791,Z 483.789,A -85,B 0,C 180,E1 10779.609,E2 10779.609} C_VEL
LIN {X 0,Y 292.651,Z 491.334,A -85,B 0,C 180,E1 10776.751,E2 10776.751} C_VEL
LIN {X 0,Y 295.716,Z 497.008,A -85,B 0,C 180,E1 10775.098,E2 10775.098} C_VEL
LIN {X 0,Y 301.411,Z 509.175,A -85,B 0,C 180,E1 10772.267,E2 10772.267} C_VEL
LIN {X 0,Y 303.278,Z 513.774,A -85,B 0,C 180,E1 10771.387,E2 10771.387} C_VEL
LIN {X 0,Y 293.154,Z 642.665,A -85,B 0,C 180,E1 10768.583,E2 10768.583} C_VEL
LIN {X 0,Y 291.489,Z 655.403,A -85,B 0,C 180,E1 10768.214,E2 10768.214} C_VEL
LIN {X 0,Y 289.727,Z 662.949,A -85,B 0,C 180,E1 10768.152,E2 10768.152} C_VEL
LIN {X 0,Y 282.924,Z 680.676,A -85,B 0,C 180,E1 10768.384,E2 10768.384} C_VEL
LIN {X 0,Y 280.542,Z 688.014,A -85,B 0,C 180,E1 10768.21,E2 10768.21} C_VEL
LIN {X 0,Y 280.278,Z 689.063,A -85,B 0,C 180,E1 10768.159,E2 10768.159} C_VEL
LIN {X 0,Y 274.473,Z 708.629,A -85,B 0,C 180,E1 10766.911,E2 10766.911} C_VEL
LIN {X 0,Y 268.937,Z 724.484,A -85,B 0,C 180,E1 10765.622,E2 10765.622} C_VEL
LIN {X 0,Y 261.932,Z 742.102,A -85,B 0,C 180,E1 10763.835,E2 10763.835} C_VEL
LIN {X 0,Y 254.251,Z 758.699,A -85,B 0,C 180,E1 10761.677,E2 10761.677} C_VEL
LIN {X 0,Y 247.273,Z 772.436,A -85,B 0,C 180,E1 10759.479,E2 10759.479} C_VEL
LIN {X 0,Y 239.337,Z 786.961,A -85,B 0,C 180,E1 10756.626,E2 10756.626} C_VEL
LIN {X 0,Y 231.031,Z 800.864,A -85,B 0,C 180,E1 10753.139,E2 10753.139} C_VEL
LIN {X 0,Y 224.5,Z 811.361,A -85,B 0,C 180,E1 10749.89,E2 10749.89} C_VEL
LIN {X 0,Y 217.572,Z 822.353,A -85,B 0,C 180,E1 10745.705,E2 10745.705} C_VEL
LIN {X 0,Y 211.485,Z 831.881,A -85,B 0,C 180,E1 10741.018,E2 10741.018} C_VEL
LIN {X 0,Y 207.202,Z 838.939,A -85,B 0,C 180,E1 10736.664,E2 10736.664} C_VEL
LIN {X 0,Y 203.661,Z 845.435,A -85,B 0,C 180,E1 10731.604,E2 10731.604} C_VEL
LIN {X 0,Y 201.136,Z 851.07,A -85,B 0,C 180,E1 10725.571,E2 10725.571} C_VEL
LIN {X 0,Y 200.208,Z 854.244,A -85,B 0,C 180,E1 10720.648,E2 10720.648} C_VEL
LIN {X 0,Y 199.976,Z 856.152,A -85,B 0,C 180,E1 10716.027,E2 10716.027} C_VEL
LIN {X 0,Y 200.006,Z 856.984,A -85,B 0,C 180,E1 10711.719,E2 10711.719} C_VEL
LIN {X 0,Y 199.997,Z 856.924,A -85,B 0,C 180,E1 10707.708,E2 10707.708} C_VEL
LIN {X 0,Y 199.983,Z 855.971,A -85,B 0,C 180,E1 10703.397,E2 10703.397} C_VEL
LIN {X 0,Y 200.308,Z 853.792,A -85,B 0,C 180,E1 10698.483,E2 10698.483} C_VEL
LIN {X 0,Y 201.799,Z 849.42,A -85,B 0,C 180,E1 10692.408,E2 10692.408} C_VEL
LIN {X 0,Y 204.332,Z 844.088,A -85,B 0,C 180,E1 10687.259,E2 10687.259} C_VEL
LIN {X 0,Y 207.925,Z 837.732,A -85,B 0,C 180,E1 10682.508,E2 10682.508} C_VEL
LIN {X 0,Y 214.025,Z 827.845,A -85,B 0,C 180,E1 10676.868,E2 10676.868} C_VEL
LIN {X 0,Y 219.884,Z 818.625,A -85,B 0,C 180,E1 10672.788,E2 10672.788} C_VEL
LIN {X 0,Y 226.753,Z 807.84,A -85,B 0,C 180,E1 10668.929,E2 10668.929} C_VEL
LIN {X 0,Y 235.071,Z 794.161,A -85,B 0,C 180,E1 10665.086,E2 10665.086} C_VEL
LIN {X 0,Y 242.17,Z 781.829,A -85,B 0,C 180,E1 10662.308,E2 10662.308} C_VEL
LIN {X 0,Y 249.968,Z 767.381,A -85,B 0,C 180,E1 10659.649,E2 10659.649} C_VEL
LIN {X 0,Y 258.231,Z 750.245,A -85,B 0,C 180,E1 10657.168,E2 10657.168} C_VEL
LIN {X 0,Y 264.559,Z 735.65,A -85,B 0,C 180,E1 10655.47,E2 10655.47} C_VEL
LIN {X 0,Y 271.235,Z 718.315,A -85,B 0,C 180,E1 10653.832,E2 10653.832} C_VEL
LIN {X 0,Y 277.296,Z 699.523,A -85,B 0,C 180,E1 10652.465,E2 10652.465} C_VEL
LIN {X 0,Y 281.788,Z 682.792,A -85,B 0,C 180,E1 10651.521,E2 10651.521} C_VEL
LIN {X 0,Y 285.774,Z 664.502,A -85,B 0,C 180,E1 10650.737,E2 10650.737} C_VEL
LIN {X 0,Y 289.019,Z 642.701,A -85,B 0,C 180,E1 10650.067,E2 10650.067} C_VEL
LIN {X 0,Y 297.145,Z 542.902,A -85,B 0,C 180,E1 10647.886,E2 10647.886} C_VEL
LIN {X 0,Y 299.168,Z 517.173,A -85,B 0,C 180,E1 10647.322,E2 10647.322} C_VEL
LIN {X 0,Y 293.854,Z 505.197,A -85,B 0,C 180,E1 10644.587,E2 10644.587} C_VEL
LIN {X 0,Y 290.465,Z 498.491,A -85,B 0,C 180,E1 10642.684,E2 10642.684} C_VEL
LIN {X 0,Y 285.682,Z 490.813,A -85,B 0,C 180,E1 10639.747,E2 10639.747} C_VEL
LIN {X 0,Y 281.032,Z 483.694,A -85,B 0,C 180,E1 10636.332,E2 10636.332} C_VEL
LIN {X 0,Y 278.022,Z 479.253,A -85,B 0,C 180,E1 10633.633,E2 10633.633} C_VEL
LIN {X 0,Y 275.17,Z 474.815,A -85,B 0,C 180,E1 10630.37,E2 10630.37} C_VEL
LIN {X 0,Y 272.138,Z 470.815,A -85,B 0,C 180,E1 10625.068,E2 10625.068} C_VEL
LIN {X 0,Y 271.653,Z 469.226,A -85,B 0,C 180,E1 10623.174,E2 10623.174} C_VEL
LIN {X 0,Y 271.554,Z 469.11,A -85,B 0,C 180,E1 10616.843,E2 10616.843} C_VEL
LIN {X 0,Y 271.899,Z 469.967,A -85,B 0,C 180,E1 10615.369,E2 10615.369} C_VEL
LIN {X 0,Y 274.302,Z 474.022,A -85,B 0,C 180,E1 10610.357,E2 10610.357} C_VEL
LIN {X 0,Y 275.311,Z 475.111,A -85,B 0,C 180,E1 10609.018,E2 10609.018} C_VEL
LIN {X 0,Y 278.12,Z 479.341,A -85,B 0,C 180,E1 10605.86,E2 10605.86} C_VEL
LIN {X 0,Y 282.391,Z 485.778,A -85,B 0,C 180,E1 10602.176,E2 10602.176} C_VEL
LIN {X 0,Y 285.881,Z 491.206,A -85,B 0,C 180,E1 10599.699,E2 10599.699} C_VEL
LIN {X 0,Y 294.899,Z 502.34,A -85,B 0,C 180,E1 10594.721,E2 10594.721} C_VEL
LIN {X 0,Y 304.133,Z 510.685,A -85,B 0,C 180,E1 10590.789,E2 10590.789} C_VEL
LIN {X 0,Y 308.451,Z 514.1,A -85,B 0,C 180,E1 10588.987,E2 10588.987} C_VEL
LIN {X 0,Y 314.145,Z 518.861,A -85,B 0,C 180,E1 10586.384,E2 10586.384} C_VEL
LIN {X 0,Y 317.043,Z 521.181,A -85,B 0,C 180,E1 10584.985,E2 10584.985} C_VEL
LIN {X 0,Y 321.766,Z 525.553,A -85,B 0,C 180,E1 10582.492,E2 10582.492} C_VEL
LIN {X 0,Y 325.362,Z 528.644,A -85,B 0,C 180,E1 10580.396,E2 10580.396} C_VEL
LIN {X 0,Y 330.319,Z 533.568,A -85,B 0,C 180,E1 10577.352,E2 10577.352} C_VEL
LIN {X 0,Y 333.386,Z 536.165,A -85,B 0,C 180,E1 10575.444,E2 10575.444} C_VEL
LIN {X 0,Y 337.826,Z 540.586,A -85,B 0,C 180,E1 10572.542,E2 10572.542} C_VEL
LIN {X 0,Y 341.503,Z 543.53,A -85,B 0,C 180,E1 10570.098,E2 10570.098} C_VEL
LIN {X 0,Y 345.902,Z 547.977,A -85,B 0,C 180,E1 10566.958,E2 10566.958} C_VEL
LIN {X 0,Y 349.99,Z 551.034,A -85,B 0,C 180,E1 10563.951,E2 10563.951} C_VEL
LIN {X 0,Y 353.522,Z 554.825,A -85,B 0,C 180,E1 10561.043,E2 10561.043} C_VEL
LIN {X 0,Y 357.228,Z 557.587,A -85,B 0,C 180,E1 10557.866,E2 10557.866} C_VEL
LIN {X 0,Y 358.945,Z 558.795,A -85,B 0,C 180,E1 10556.288,E2 10556.288} C_VEL
LIN {X 0,Y 362.027,Z 562.327,A -85,B 0,C 180,E1 10553.09,E2 10553.09} C_VEL
LIN {X 0,Y 365.031,Z 564.683,A -85,B 0,C 180,E1 10549.688,E2 10549.688} C_VEL
LIN {X 0,Y 367.681,Z 565.964,A -85,B 0,C 180,E1 10546.265,E2 10546.265} C_VEL
LIN {X 0,Y 368.828,Z 567.094,A -85,B 0,C 180,E1 10544.442,E2 10544.442} C_VEL
LIN {X 0,Y 370.373,Z 569.293,A -85,B 0,C 180,E1 10541.365,E2 10541.365} C_VEL
LIN {X 0,Y 371.681,Z 570.653,A -85,B 0,C 180,E1 10538.197,E2 10538.197} C_VEL
LIN {X 0,Y 372.552,Z 571.446,A -85,B 0,C 180,E1 10534.927,E2 10534.927} C_VEL
LIN {X 0,Y 373.034,Z 571.809,A -85,B 0,C 180,E1 10531.536,E2 10531.536} C_VEL
LIN {X 0,Y 373.039,Z 571.807,A -85,B 0,C 180,E1 10528.157,E2 10528.157} C_VEL
LIN {X 0,Y 372.468,Z 571.383,A -85,B 0,C 180,E1 10524.702,E2 10524.702} C_VEL
LIN {X 0,Y 371.433,Z 570.45,A -85,B 0,C 180,E1 10521.174,E2 10521.174} C_VEL
LIN {X 0,Y 370.012,Z 568.858,A -85,B 0,C 180,E1 10517.833,E2 10517.833} C_VEL
LIN {X 0,Y 368.124,Z 566.162,A -85,B 0,C 180,E1 10514.402,E2 10514.402} C_VEL
LIN {X 0,Y 365.584,Z 565.008,A -85,B 0,C 180,E1 10511.007,E2 10511.007} C_VEL
LIN {X 0,Y 362.836,Z 563.042,A -85,B 0,C 180,E1 10507.777,E2 10507.777} C_VEL
LIN {X 0,Y 359.921,Z 560.025,A -85,B 0,C 180,E1 10504.672,E2 10504.672} C_VEL
LIN {X 0,Y 358.147,Z 558.039,A -85,B 0,C 180,E1 10502.921,E2 10502.921} C_VEL
LIN {X 0,Y 354.611,Z 555.767,A -85,B 0,C 180,E1 10499.876,E2 10499.876} C_VEL
LIN {X 0,Y 350.936,Z 552.213,A -85,B 0,C 180,E1 10496.838,E2 10496.838} C_VEL
LIN {X 0,Y 348.983,Z 550.161,A -85,B 0,C 180,E1 10495.295,E2 10495.295} C_VEL
LIN {X 0,Y 344.829,Z 547.03,A -85,B 0,C 180,E1 10492.281,E2 10492.281} C_VEL
LIN {X 0,Y 340.223,Z 542.356,A -85,B 0,C 180,E1 10489.034,E2 10489.034} C_VEL
LIN {X 0,Y 335.613,Z 538.578,A -85,B 0,C 180,E1 10486.009,E2 10486.009} C_VEL
LIN {X 0,Y 331.875,Z 534.738,A -85,B 0,C 180,E1 10483.609,E2 10483.609} C_VEL
LIN {X 0,Y 327.193,Z 530.655,A -85,B 0,C 180,E1 10480.727,E2 10480.727} C_VEL
LIN {X 0,Y 323.675,Z 527.06,A -85,B 0,C 180,E1 10478.595,E2 10478.595} C_VEL
LIN {X 0,Y 318.745,Z 522.917,A -85,B 0,C 180,E1 10475.903,E2 10475.903} C_VEL
LIN {X 0,Y 315.254,Z 519.631,A -85,B 0,C 180,E1 10474.131,E2 10474.131} C_VEL
LIN {X 0,Y 309.976,Z 515.525,A -85,B 0,C 180,E1 10471.708,E2 10471.708} C_VEL
LIN {X 0,Y 305.189,Z 511.434,A -85,B 0,C 180,E1 10469.639,E2 10469.639} C_VEL
LIN {X 0,Y 298.237,Z 505.644,A -85,B 0,C 180,E1 10466.791,E2 10466.791} C_VEL
LIN {X 0,Y 289.977,Z 496.726,A -85,B 0,C 180,E1 10462.76,E2 10462.76} C_VEL
LIN {X 0,Y 281.65,Z 484.472,A -85,B 0,C 180,E1 10457.232,E2 10457.232} C_VEL
LIN {X 0,Y 277.907,Z 479.124,A -85,B 0,C 180,E1 10453.938,E2 10453.938} C_VEL
LIN {X 0,Y 274.926,Z 474.514,A -85,B 0,C 180,E1 10450.467,E2 10450.467} C_VEL
LIN {X 0,Y 272.068,Z 470.609,A -85,B 0,C 180,E1 10445.262,E2 10445.262} C_VEL
LIN {X 0,Y 271.65,Z 469.225,A -85,B 0,C 180,E1 10443.578,E2 10443.578} C_VEL
LIN {X 0,Y 271.511,Z 469.075,A -85,B 0,C 180,E1 10437.458,E2 10437.458} C_VEL
LIN {X 0,Y 271.849,Z 469.792,A -85,B 0,C 180,E1 10435.984,E2 10435.984} C_VEL
LIN {X 0,Y 274.159,Z 473.928,A -85,B 0,C 180,E1 10430.969,E2 10430.969} C_VEL
LIN {X 0,Y 275.242,Z 474.987,A -85,B 0,C 180,E1 10429.527,E2 10429.527} C_VEL
LIN {X 0,Y 278.129,Z 479.363,A -85,B 0,C 180,E1 10426.267,E2 10426.267} C_VEL
LIN {X 0,Y 282.146,Z 485.4,A -85,B 0,C 180,E1 10422.78,E2 10422.78} C_VEL
LIN {X 0,Y 286.044,Z 491.387,A -85,B 0,C 180,E1 10420.013,E2 10420.013} C_VEL
LIN {X 0,Y 291.375,Z 500.001,A -85,B 0,C 180,E1 10416.803,E2 10416.803} C_VEL
LIN {X 0,Y 296.495,Z 510.962,A -85,B 0,C 180,E1 10414.018,E2 10414.018} C_VEL
LIN {X 0,Y 299.193,Z 517.518,A -85,B 0,C 180,E1 10412.651,E2 10412.651} C_VEL
LIN {X 0,Y 289.031,Z 642.635,A -85,B 0,C 180,E1 10409.935,E2 10409.935} C_VEL
LIN {X 0,Y 285.749,Z 664.628,A -85,B 0,C 180,E1 10409.258,E2 10409.258} C_VEL
LIN {X 0,Y 281.788,Z 682.792,A -85,B 0,C 180,E1 10408.479,E2 10408.479} C_VEL
LIN {X 0,Y 280.278,Z 689.063,A -85,B 0,C 180,E1 10408.159,E2 10408.159} C_VEL
LIN {X 0,Y 277.842,Z 696.355,A -85,B 0,C 180,E1 10407.924,E2 10407.924} C_VEL
LIN {X 0,Y 269.251,Z 713.305,A -85,B 0,C 180,E1 10407.767,E2 10407.767} C_VEL
LIN {X 0,Y 266.022,Z 720.189,A -85,B 0,C 180,E1 10407.422,E2 10407.422} C_VEL
LIN {X 0,Y 265.639,Z 721.143,A -85,B 0,C 180,E1 10407.342,E2 10407.342} C_VEL
LIN {X 0,Y 259.599,Z 736.217,A -85,B 0,C 180,E1 10405.9,E2 10405.9} C_VEL
LIN {X 0,Y 252.547,Z 751.874,A -85,B 0,C 180,E1 10404.058,E2 10404.058} C_VEL
LIN {X 0,Y 243.604,Z 769.387,A -85,B 0,C 180,E1 10401.432,E2 10401.432} C_VEL
LIN {X 0,Y 236.374,Z 782.232,A -85,B 0,C 180,E1 10399.021,E2 10399.021} C_VEL
LIN {X 0,Y 228.81,Z 794.811,A -85,B 0,C 180,E1 10396.137,E2 10396.137} C_VEL
LIN {X 0,Y 220.14,Z 808.318,A -85,B 0,C 180,E1 10392.228,E2 10392.228} C_VEL
LIN {X 0,Y 213.229,Z 818.634,A -85,B 0,C 180,E1 10388.443,E2 10388.443} C_VEL
LIN {X 0,Y 207.19,Z 827.603,A -85,B 0,C 180,E1 10384.375,E2 10384.375} C_VEL
LIN {X 0,Y 200.672,Z 837.489,A -85,B 0,C 180,E1 10378.575,E2 10378.575} C_VEL
LIN {X 0,Y 196.796,Z 843.846,A -85,B 0,C 180,E1 10373.663,E2 10373.663} C_VEL
LIN {X 0,Y 194.03,Z 849.179,A -85,B 0,C 180,E1 10368.32,E2 10368.32} C_VEL
LIN {X 0,Y 192.368,Z 853.553,A -85,B 0,C 180,E1 10361.999,E2 10361.999} C_VEL
LIN {X 0,Y 191.991,Z 855.733,A -85,B 0,C 180,E1 10356.879,E2 10356.879} C_VEL
LIN {X 0,Y 191.998,Z 856.688,A -85,B 0,C 180,E1 10352.388,E2 10352.388} C_VEL
LIN {X 0,Y 192.007,Z 856.748,A -85,B 0,C 180,E1 10348.21,E2 10348.21} C_VEL
LIN {X 0,Y 191.98,Z 855.914,A -85,B 0,C 180,E1 10343.721,E2 10343.721} C_VEL
LIN {X 0,Y 192.252,Z 854.005,A -85,B 0,C 180,E1 10338.906,E2 10338.906} C_VEL
LIN {X 0,Y 193.298,Z 850.829,A -85,B 0,C 180,E1 10333.781,E2 10333.781} C_VEL
LIN {X 0,Y 196.242,Z 844.856,A -85,B 0,C 180,E1 10327.219,E2 10327.219} C_VEL
LIN {X 0,Y 199.895,Z 838.697,A -85,B 0,C 180,E1 10322.279,E2 10322.279} C_VEL
LIN {X 0,Y 204.808,Z 831.167,A -85,B 0,C 180,E1 10317.521,E2 10317.521} C_VEL
LIN {X 0,Y 212.155,Z 820.246,A -85,B 0,C 180,E1 10312.218,E2 10312.218} C_VEL
LIN {X 0,Y 218.732,Z 810.414,A -85,B 0,C 180,E1 10308.486,E2 10308.486} C_VEL
LIN {X 0,Y 226.156,Z 799.034,A -85,B 0,C 180,E1 10304.98,E2 10304.98} C_VEL
LIN {X 0,Y 235.228,Z 784.216,A -85,B 0,C 180,E1 10301.392,E2 10301.392} C_VEL
LIN {X 0,Y 242.674,Z 771.072,A -85,B 0,C 180,E1 10298.859,E2 10298.859} C_VEL
LIN {X 0,Y 250.266,Z 756.565,A -85,B 0,C 180,E1 10296.582,E2 10296.582} C_VEL
LIN {X 0,Y 258.547,Z 738.719,A -85,B 0,C 180,E1 10294.367,E2 10294.367} C_VEL
LIN {X 0,Y 264.807,Z 723.324,A -85,B 0,C 180,E1 10292.85,E2 10292.85} C_VEL
LIN {X 0,Y 270.515,Z 707.328,A -85,B 0,C 180,E1 10291.578,E2 10291.578} C_VEL
LIN {X 0,Y 276.744,Z 686.273,A -85,B 0,C 180,E1 10290.292,E2 10290.292} C_VEL
LIN {X 0,Y 280.867,Z 668.557,A -85,B 0,C 180,E1 10289.498,E2 10289.498} C_VEL
LIN {X 0,Y 284.127,Z 650.069,A -85,B 0,C 180,E1 10288.876,E2 10288.876} C_VEL
LIN {X 0,Y 286.914,Z 622.816,A -85,B 0,C 180,E1 10288.218,E2 10288.218} C_VEL
LIN {X 0,Y 295.186,Z 520.823,A -85,B 0,C 180,E1 10285.998,E2 10285.998} C_VEL
LIN {X 0,Y 290.134,Z 509.239,A -85,B 0,C 180,E1 10283.194,E2 10283.194} C_VEL
LIN {X 0,Y 287.058,Z 503.505,A -85,B 0,C 180,E1 10281.353,E2 10281.353} C_VEL
LIN {X 0,Y 282.454,Z 495.944,A -85,B 0,C 180,E1 10278.265,E2 10278.265} C_VEL
LIN {X 0,Y 278.966,Z 490.613,A -85,B 0,C 180,E1 10275.495,E2 10275.495} C_VEL
LIN {X 0,Y 276.528,Z 486.832,A -85,B 0,C 180,E1 10273.175,E2 10273.175} C_VEL
LIN {X 0,Y 273.644,Z 482.301,A -85,B 0,C 180,E1 10269.685,E2 10269.685} C_VEL
LIN {X 0,Y 271.082,Z 478.708,A -85,B 0,C 180,E1 10264.875,E2 10264.875} C_VEL
LIN {X 0,Y 270.628,Z 477.125,A -85,B 0,C 180,E1 10262.974,E2 10262.974} C_VEL
LIN {X 0,Y 270.626,Z 477.119,A -85,B 0,C 180,E1 10256.621,E2 10256.621} C_VEL
LIN {X 0,Y 273.485,Z 482.147,A -85,B 0,C 180,E1 10250.116,E2 10250.116} C_VEL
LIN {X 0,Y 274.228,Z 483.315,A -85,B 0,C 180,E1 10249.081,E2 10249.081} C_VEL
LIN {X 0,Y 277.329,Z 488.031,A -85,B 0,C 180,E1 10245.606,E2 10245.606} C_VEL
LIN {X 0,Y 280.818,Z 493.46,A -85,B 0,C 180,E1 10242.555,E2 10242.555} C_VEL
LIN {X 0,Y 292.631,Z 509.532,A -85,B 0,C 180,E1 10235.268,E2 10235.268} C_VEL
LIN {X 0,Y 302.156,Z 518.235,A -85,B 0,C 180,E1 10231.122,E2 10231.122} C_VEL
LIN {X 0,Y 306.717,Z 521.855,A -85,B 0,C 180,E1 10229.228,E2 10229.228} C_VEL
LIN {X 0,Y 312.631,Z 526.651,A -85,B 0,C 180,E1 10226.585,E2 10226.585} C_VEL
LIN {X 0,Y 315.83,Z 529.317,A -85,B 0,C 180,E1 10225.052,E2 10225.052} C_VEL
LIN {X 0,Y 320.914,Z 533.816,A -85,B 0,C 180,E1 10222.375,E2 10222.375} C_VEL
LIN {X 0,Y 323.903,Z 536.419,A -85,B 0,C 180,E1 10220.641,E2 10220.641} C_VEL
LIN {X 0,Y 328.92,Z 541.343,A -85,B 0,C 180,E1 10217.572,E2 10217.572} C_VEL
LIN {X 0,Y 331.802,Z 543.742,A -85,B 0,C 180,E1 10215.791,E2 10215.791} C_VEL
LIN {X 0,Y 336.425,Z 548.333,A -85,B 0,C 180,E1 10212.785,E2 10212.785} C_VEL
LIN {X 0,Y 340.133,Z 551.279,A -85,B 0,C 180,E1 10210.346,E2 10210.346} C_VEL
LIN {X 0,Y 344.691,Z 555.841,A -85,B 0,C 180,E1 10207.106,E2 10207.106} C_VEL
LIN {X 0,Y 348.794,Z 558.963,A -85,B 0,C 180,E1 10204.079,E2 10204.079} C_VEL
LIN {X 0,Y 352.474,Z 562.811,A -85,B 0,C 180,E1 10201.075,E2 10201.075} C_VEL
LIN {X 0,Y 356.121,Z 565.488,A -85,B 0,C 180,E1 10197.96,E2 10197.96} C_VEL
LIN {X 0,Y 357.728,Z 566.596,A -85,B 0,C 180,E1 10196.497,E2 10196.497} C_VEL
LIN {X 0,Y 360.701,Z 569.994,A -85,B 0,C 180,E1 10193.46,E2 10193.46} C_VEL
LIN {X 0,Y 363.563,Z 572.319,A -85,B 0,C 180,E1 10190.274,E2 10190.274} C_VEL
LIN {X 0,Y 366.279,Z 573.762,A -85,B 0,C 180,E1 10186.819,E2 10186.819} C_VEL
LIN {X 0,Y 367.504,Z 574.624,A -85,B 0,C 180,E1 10184.978,E2 10184.978} C_VEL
LIN {X 0,Y 369.242,Z 577.076,A -85,B 0,C 180,E1 10181.717,E2 10181.717} C_VEL
LIN {X 0,Y 370.57,Z 578.478,A -85,B 0,C 180,E1 10178.534,E2 10178.534} C_VEL
LIN {X 0,Y 371.535,Z 579.36,A -85,B 0,C 180,E1 10175.095,E2 10175.095} C_VEL
LIN {X 0,Y 372.06,Z 579.752,A -85,B 0,C 180,E1 10171.694,E2 10171.694} C_VEL
LIN {X 0,Y 372.06,Z 579.753,A -85,B 0,C 180,E1 10168.306,E2 10168.306} C_VEL
LIN {X 0,Y 371.535,Z 579.36,A -85,B 0,C 180,E1 10164.905,E2 10164.905} C_VEL
LIN {X 0,Y 370.571,Z 578.477,A -85,B 0,C 180,E1 10161.466,E2 10161.466} C_VEL
LIN {X 0,Y 369.242,Z 577.077,A -85,B 0,C 180,E1 10158.283,E2 10158.283} C_VEL
LIN {X 0,Y 367.467,Z 574.571,A -85,B 0,C 180,E1 10154.961,E2 10154.961} C_VEL
LIN {X 0,Y 366.02,Z 573.665,A -85,B 0,C 180,E1 10152.842,E2 10152.842} C_VEL
LIN {X 0,Y 363.235,Z 572.103,A -85,B 0,C 180,E1 10149.37,E2 10149.37} C_VEL
LIN {X 0,Y 360.292,Z 569.581,A -85,B 0,C 180,E1 10146.099,E2 10146.099} C_VEL
LIN {X 0,Y 357.076,Z 565.953,A -85,B 0,C 180,E1 10142.844,E2 10142.844} C_VEL
LIN {X 0,Y 353.487,Z 563.669,A -85,B 0,C 180,E1 10139.77,E2 10139.77} C_VEL
LIN {X 0,Y 349.759,Z 560.129,A -85,B 0,C 180,E1 10136.712,E2 10136.712} C_VEL
LIN {X 0,Y 347.625,Z 557.934,A -85,B 0,C 180,E1 10135.04,E2 10135.04} C_VEL
LIN {X 0,Y 343.495,Z 554.806,A -85,B 0,C 180,E1 10132.06,E2 10132.06} C_VEL
LIN {X 0,Y 338.832,Z 550.115,A -85,B 0,C 180,E1 10128.79,E2 10128.79} C_VEL
LIN {X 0,Y 334.205,Z 546.327,A -85,B 0,C 180,E1 10125.766,E2 10125.766} C_VEL
LIN {X 0,Y 330.298,Z 542.383,A -85,B 0,C 180,E1 10123.272,E2 10123.272} C_VEL
LIN {X 0,Y 325.406,Z 538.076,A -85,B 0,C 180,E1 10120.287,E2 10120.287} C_VEL
LIN {X 0,Y 322.171,Z 534.799,A -85,B 0,C 180,E1 10118.354,E2 10118.354} C_VEL
LIN {X 0,Y 317.34,Z 530.829,A -85,B 0,C 180,E1 10115.752,E2 10115.752} C_VEL
LIN {X 0,Y 313.27,Z 527.109,A -85,B 0,C 180,E1 10113.723,E2 10113.723} C_VEL
LIN {X 0,Y 307.338,Z 522.401,A -85,B 0,C 180,E1 10111.029,E2 10111.029} C_VEL
LIN {X 0,Y 302.803,Z 518.693,A -85,B 0,C 180,E1 10109.135,E2 10109.135} C_VEL
LIN {X 0,Y 295.508,Z 512.38,A -85,B 0,C 180,E1 10106.083,E2 10106.083} C_VEL
LIN {X 0,Y 288.002,Z 504.102,A -85,B 0,C 180,E1 10102.278,E2 10102.278} C_VEL
LIN {X 0,Y 279.916,Z 491.88,A -85,B 0,C 180,E1 10096.701,E2 10096.701} C_VEL
LIN {X 0,Y 276.521,Z 486.818,A -85,B 0,C 180,E1 10093.583,E2 10093.583} C_VEL
LIN {X 0,Y 273.64,Z 482.271,A -85,B 0,C 180,E1 10090.091,E2 10090.091} C_VEL
LIN {X 0,Y 270.93,Z 478.203,A -85,B 0,C 180,E1 10084.753,E2 10084.753} C_VEL
LIN {X 0,Y 270.626,Z 477.12,A -85,B 0,C 180,E1 10083.379,E2 10083.379} C_VEL
LIN {X 0,Y 270.628,Z 477.124,A -85,B 0,C 180,E1 10077.026,E2 10077.026} C_VEL
LIN {X 0,Y 273.189,Z 481.935,A -85,B 0,C 180,E1 10070.937,E2 10070.937} C_VEL
LIN {X 0,Y 274.016,Z 482.866,A -85,B 0,C 180,E1 10069.798,E2 10069.798} C_VEL
LIN {X 0,Y 277.546,Z 488.357,A -85,B 0,C 180,E1 10065.812,E2 10065.812} C_VEL
LIN {X 0,Y 280.699,Z 493.298,A -85,B 0,C 180,E1 10063.062,E2 10063.062} C_VEL
LIN {X 0,Y 284.241,Z 498.867,A -85,B 0,C 180,E1 10060.47,E2 10060.47} C_VEL
LIN {X 0,Y 289.044,Z 506.935,A -85,B 0,C 180,E1 10057.455,E2 10057.455} C_VEL
LIN {X 0,Y 293.76,Z 517.476,A -85,B 0,C 180,E1 10054.759,E2 10054.759} C_VEL
LIN {X 0,Y 295.25,Z 521.362,A -85,B 0,C 180,E1 10053.948,E2 10053.948} C_VEL
LIN {X 0,Y 285.095,Z 642.408,A -85,B 0,C 180,E1 10051.331,E2 10051.331} C_VEL
LIN {X 0,Y 281.7,Z 664.538,A -85,B 0,C 180,E1 10050.656,E2 10050.656} C_VEL
LIN {X 0,Y 277.67,Z 682.555,A -85,B 0,C 180,E1 10049.893,E2 10049.893} C_VEL
LIN {X 0,Y 272.858,Z 699.97,A -85,B 0,C 180,E1 10048.919,E2 10048.919} C_VEL
LIN {X 0,Y 265.863,Z 720.559,A -85,B 0,C 180,E1 10047.394,E2 10047.394} C_VEL
LIN {X 0,Y 265.639,Z 721.143,A -85,B 0,C 180,E1 10047.342,E2 10047.342} C_VEL
LIN {X 0,Y 262.419,Z 728.177,A -85,B 0,C 180,E1 10046.901,E2 10046.901} C_VEL
LIN {X 0,Y 251.713,Z 744.864,A -85,B 0,C 180,E1 10046.236,E2 10046.236} C_VEL
LIN {X 0,Y 248.141,Z 751.061,A -85,B 0,C 180,E1 10045.65,E2 10045.65} C_VEL
LIN {X 0,Y 238.933,Z 768.584,A -85,B 0,C 180,E1 10043.059,E2 10043.059} C_VEL
LIN {X 0,Y 231.112,Z 781.972,A -85,B 0,C 180,E1 10040.554,E2 10040.554} C_VEL
LIN {X 0,Y 223.219,Z 794.57,A -85,B 0,C 180,E1 10037.651,E2 10037.651} C_VEL
LIN {X 0,Y 213.735,Z 808.637,A -85,B 0,C 180,E1 10033.511,E2 10033.511} C_VEL
LIN {X 0,Y 206.595,Z 818.761,A -85,B 0,C 180,E1 10029.704,E2 10029.704} C_VEL
LIN {X 0,Y 199.714,Z 828.448,A -85,B 0,C 180,E1 10025.15,E2 10025.15} C_VEL
LIN {X 0,Y 193.495,Z 837.246,A -85,B 0,C 180,E1 10019.739,E2 10019.739} C_VEL
LIN {X 0,Y 189.314,Z 843.604,A -85,B 0,C 180,E1 10014.659,E2 10014.659} C_VEL
LIN {X 0,Y 186.292,Z 848.938,A -85,B 0,C 180,E1 10009.11,E2 10009.11} C_VEL
LIN {X 0,Y 184.44,Z 853.313,A -85,B 0,C 180,E1 10002.523,E2 10002.523} C_VEL
LIN {X 0,Y 184.003,Z 855.495,A -85,B 0,C 180,E1 9997.179,E2 9997.179} C_VEL
LIN {X 0,Y 184.001,Z 856.451,A -85,B 0,C 180,E1 9992.491,E2 9992.491} C_VEL
LIN {X 0,Y 184.009,Z 856.512,A -85,B 0,C 180,E1 9988.132,E2 9988.132} C_VEL
LIN {X 0,Y 183.985,Z 855.676,A -85,B 0,C 180,E1 9983.447,E2 9983.447} C_VEL
LIN {X 0,Y 184.305,Z 853.765,A -85,B 0,C 180,E1 9978.421,E2 9978.421} C_VEL
LIN {X 0,Y 185.483,Z 850.588,A -85,B 0,C 180,E1 9973.077,E2 9973.077} C_VEL
LIN {X 0,Y 188.711,Z 844.614,A -85,B 0,C 180,E1 9966.255,E2 9966.255} C_VEL
LIN {X 0,Y 192.662,Z 838.454,A -85,B 0,C 180,E1 9961.143,E2 9961.143} C_VEL
LIN {X 0,Y 197.922,Z 830.924,A -85,B 0,C 180,E1 9956.243,E2 9956.243} C_VEL
LIN {X 0,Y 205.723,Z 820.004,A -85,B 0,C 180,E1 9950.816,E2 9950.816} C_VEL
LIN {X 0,Y 212.655,Z 810.172,A -85,B 0,C 180,E1 9947.02,E2 9947.02} C_VEL
LIN {X 0,Y 220.442,Z 798.792,A -85,B 0,C 180,E1 9943.474,E2 9943.474} C_VEL
LIN {X 0,Y 229.883,Z 784.018,A -85,B 0,C 180,E1 9939.874,E2 9939.874} C_VEL
LIN {X 0,Y 237.648,Z 770.831,A -85,B 0,C 180,E1 9937.33,E2 9937.33} C_VEL
LIN {X 0,Y 245.811,Z 755.757,A -85,B 0,C 180,E1 9934.976,E2 9934.976} C_VEL
LIN {X 0,Y 254.096,Z 738.399,A -85,B 0,C 180,E1 9932.85,E2 9932.85} C_VEL
LIN {X 0,Y 260.511,Z 723.085,A -85,B 0,C 180,E1 9931.357,E2 9931.357} C_VEL
LIN {X 0,Y 266.381,Z 707.089,A -85,B 0,C 180,E1 9930.1,E2 9930.1} C_VEL
LIN {X 0,Y 272.775,Z 686.036,A -85,B 0,C 180,E1 9928.833,E2 9928.833} C_VEL
LIN {X 0,Y 277.001,Z 668.32,A -85,B 0,C 180,E1 9928.053,E2 9928.053} C_VEL
LIN {X 0,Y 280.34,Z 649.832,A -85,B 0,C 180,E1 9927.44,E2 9927.44} C_VEL
LIN {X 0,Y 283.207,Z 622.579,A -85,B 0,C 180,E1 9926.787,E2 9926.787} C_VEL
LIN {X 0,Y 291.403,Z 524.805,A -85,B 0,C 180,E1 9924.673,E2 9924.673} C_VEL
LIN {X 0,Y 287.177,Z 514.831,A -85,B 0,C 180,E1 9922.154,E2 9922.154} C_VEL
LIN {X 0,Y 283.795,Z 508.635,A -85,B 0,C 180,E1 9919.991,E2 9919.991} C_VEL
LIN {X 0,Y 280.134,Z 502.563,A -85,B 0,C 180,E1 9917.347,E2 9917.347} C_VEL
LIN {X 0,Y 277.406,Z 498.154,A -85,B 0,C 180,E1 9915.049,E2 9915.049} C_VEL
LIN {X 0,Y 275.053,Z 494.408,A -85,B 0,C 180,E1 9912.713,E2 9912.713} C_VEL
LIN {X 0,Y 272.367,Z 490.061,A -85,B 0,C 180,E1 9909.304,E2 9909.304} C_VEL
LIN {X 0,Y 269.913,Z 486.219,A -85,B 0,C 180,E1 9904.258,E2 9904.258} C_VEL
LIN {X 0,Y 269.605,Z 485.024,A -85,B 0,C 180,E1 9902.772,E2 9902.772} C_VEL
LIN {X 0,Y 269.651,Z 485.075,A -85,B 0,C 180,E1 9896.608,E2 9896.608} C_VEL
LIN {X 0,Y 272.072,Z 489.779,A -85,B 0,C 180,E1 9890.704,E2 9890.704} C_VEL
LIN {X 0,Y 272.795,Z 490.699,A -85,B 0,C 180,E1 9889.664,E2 9889.664} C_VEL
LIN {X 0,Y 275.923,Z 495.775,A -85,B 0,C 180,E1 9885.959,E2 9885.959} C_VEL
LIN {X 0,Y 279.138,Z 500.928,A -85,B 0,C 180,E1 9883.037,E2 9883.037} C_VEL
LIN {X 0,Y 290.574,Z 516.9,A -85,B 0,C 180,E1 9875.731,E2 9875.731} C_VEL
LIN {X 0,Y 300.19,Z 525.784,A -85,B 0,C 180,E1 9871.459,E2 9871.459} C_VEL
LIN {X 0,Y 304.582,Z 529.239,A -85,B 0,C 180,E1 9869.645,E2 9869.645} C_VEL
LIN {X 0,Y 310.357,Z 533.901,A -85,B 0,C 180,E1 9867.135,E2 9867.135} C_VEL
LIN {X 0,Y 314.064,Z 536.91,A -85,B 0,C 180,E1 9865.383,E2 9865.383} C_VEL
LIN {X 0,Y 319.376,Z 541.552,A -85,B 0,C 180,E1 9862.615,E2 9862.615} C_VEL
LIN {X 0,Y 322.604,Z 544.373,A -85,B 0,C 180,E1 9860.788,E2 9860.788} C_VEL
LIN {X 0,Y 327.634,Z 549.21,A -85,B 0,C 180,E1 9857.722,E2 9857.722} C_VEL
LIN {X 0,Y 330.363,Z 551.51,A -85,B 0,C 180,E1 9856.032,E2 9856.032} C_VEL
LIN {X 0,Y 335.021,Z 556.079,A -85,B 0,C 180,E1 9853.029,E2 9853.029} C_VEL
LIN {X 0,Y 338.794,Z 559.105,A -85,B 0,C 180,E1 9850.544,E2 9850.544} C_VEL
LIN {X 0,Y 343.31,Z 563.584,A -85,B 0,C 180,E1 9847.354,E2 9847.354} C_VEL
LIN {X 0,Y 347.437,Z 566.693,A -85,B 0,C 180,E1 9844.335,E2 9844.335} C_VEL
LIN {X 0,Y 351.136,Z 570.543,A -85,B 0,C 180,E1 9841.344,E2 9841.344} C_VEL
LIN {X 0,Y 354.894,Z 573.323,A -85,B 0,C 180,E1 9838.159,E2 9838.159} C_VEL
LIN {X 0,Y 356.623,Z 574.546,A -85,B 0,C 180,E1 9836.596,E2 9836.596} C_VEL
LIN {X 0,Y 359.685,Z 577.968,A -85,B 0,C 180,E1 9833.487,E2 9833.487} C_VEL
LIN {X 0,Y 362.675,Z 580.345,A -85,B 0,C 180,E1 9830.157,E2 9830.157} C_VEL
LIN {X 0,Y 365.391,Z 581.737,A -85,B 0,C 180,E1 9826.697,E2 9826.697} C_VEL
LIN {X 0,Y 366.488,Z 582.587,A -85,B 0,C 180,E1 9825.021,E2 9825.021} C_VEL
LIN {X 0,Y 368.247,Z 585.019,A -85,B 0,C 180,E1 9821.749,E2 9821.749} C_VEL
LIN {X 0,Y 369.584,Z 586.419,A -85,B 0,C 180,E1 9818.557,E2 9818.557} C_VEL
LIN {X 0,Y 370.554,Z 587.3,A -85,B 0,C 180,E1 9815.108,E2 9815.108} C_VEL
LIN {X 0,Y 371.084,Z 587.692,A -85,B 0,C 180,E1 9811.698,E2 9811.698} C_VEL
LIN {X 0,Y 371.082,Z 587.691,A -85,B 0,C 180,E1 9808.456,E2 9808.456} C_VEL
LIN {X 0,Y 370.591,Z 587.325,A -85,B 0,C 180,E1 9805.047,E2 9805.047} C_VEL
LIN {X 0,Y 369.704,Z 586.534,A -85,B 0,C 180,E1 9801.75,E2 9801.75} C_VEL
LIN {X 0,Y 368.382,Z 585.177,A -85,B 0,C 180,E1 9798.572,E2 9798.572} C_VEL
LIN {X 0,Y 366.742,Z 582.943,A -85,B 0,C 180,E1 9795.388,E2 9795.388} C_VEL
LIN {X 0,Y 365.646,Z 581.825,A -85,B 0,C 180,E1 9793.642,E2 9793.642} C_VEL
LIN {X 0,Y 362.961,Z 580.533,A -85,B 0,C 180,E1 9790.195,E2 9790.195} C_VEL
LIN {X 0,Y 359.953,Z 578.231,A -85,B 0,C 180,E1 9786.816,E2 9786.816} C_VEL
LIN {X 0,Y 356.893,Z 574.903,A -85,B 0,C 180,E1 9783.678,E2 9783.678} C_VEL
LIN {X 0,Y 355.729,Z 573.74,A -85,B 0,C 180,E1 9782.552,E2 9782.552} C_VEL
LIN {X 0,Y 352.127,Z 571.367,A -85,B 0,C 180,E1 9779.453,E2 9779.453} C_VEL
LIN {X 0,Y 348.292,Z 567.697,A -85,B 0,C 180,E1 9776.339,E2 9776.339} C_VEL
LIN {X 0,Y 346.505,Z 565.844,A -85,B 0,C 180,E1 9774.956,E2 9774.956} C_VEL
LIN {X 0,Y 342.327,Z 562.734,A -85,B 0,C 180,E1 9771.956,E2 9771.956} C_VEL
LIN {X 0,Y 337.441,Z 557.873,A -85,B 0,C 180,E1 9768.545,E2 9768.545} C_VEL
LIN {X 0,Y 332.616,Z 553.914,A -85,B 0,C 180,E1 9765.418,E2 9765.418} C_VEL
LIN {X 0,Y 328.879,Z 550.132,A -85,B 0,C 180,E1 9763.027,E2 9763.027} C_VEL
LIN {X 0,Y 323.982,Z 545.869,A -85,B 0,C 180,E1 9760.062,E2 9760.062} C_VEL
LIN {X 0,Y 320.385,Z 542.302,A -85,B 0,C 180,E1 9757.924,E2 9757.924} C_VEL
LIN {X 0,Y 315.276,Z 538.1,A -85,B 0,C 180,E1 9755.241,E2 9755.241} C_VEL
LIN {X 0,Y 311.312,Z 534.575,A -85,B 0,C 180,E1 9753.301,E2 9753.301} C_VEL
LIN {X 0,Y 305.193,Z 529.787,A -85,B 0,C 180,E1 9750.615,E2 9750.615} C_VEL
LIN {X 0,Y 301.043,Z 526.394,A -85,B 0,C 180,E1 9748.886,E2 9748.886} C_VEL
LIN {X 0,Y 293.588,Z 519.954,A -85,B 0,C 180,E1 9745.724,E2 9745.724} C_VEL
LIN {X 0,Y 285.969,Z 511.362,A -85,B 0,C 180,E1 9741.743,E2 9741.743} C_VEL
LIN {X 0,Y 278.206,Z 499.283,A -85,B 0,C 180,E1 9736.162,E2 9736.162} C_VEL
LIN {X 0,Y 274.949,Z 494.284,A -85,B 0,C 180,E1 9733.02,E2 9733.02} C_VEL
LIN {X 0,Y 272.365,Z 490.026,A -85,B 0,C 180,E1 9729.712,E2 9729.712} C_VEL
LIN {X 0,Y 269.837,Z 485.9,A -85,B 0,C 180,E1 9724.347,E2 9724.347} C_VEL
LIN {X 0,Y 269.604,Z 485.017,A -85,B 0,C 180,E1 9723.179,E2 9723.179} C_VEL
LIN {X 0,Y 269.653,Z 485.076,A -85,B 0,C 180,E1 9717.015,E2 9717.015} C_VEL
LIN {X 0,Y 271.933,Z 489.684,A -85,B 0,C 180,E1 9711.321,E2 9711.321} C_VEL
LIN {X 0,Y 272.797,Z 490.733,A -85,B 0,C 180,E1 9710.072,E2 9710.072} C_VEL
LIN {X 0,Y 276.035,Z 495.905,A -85,B 0,C 180,E1 9706.267,E2 9706.267} C_VEL
LIN {X 0,Y 279.022,Z 500.764,A -85,B 0,C 180,E1 9703.547,E2 9703.547} C_VEL
LIN {X 0,Y 283.095,Z 507.318,A -85,B 0,C 180,E1 9700.495,E2 9700.495} C_VEL
LIN {X 0,Y 287.018,Z 514.481,A -85,B 0,C 180,E1 9697.946,E2 9697.946} C_VEL
LIN {X 0,Y 291.279,Z 524.499,A -85,B 0,C 180,E1 9695.397,E2 9695.397} C_VEL
LIN {X 0,Y 291.448,Z 525.375,A -85,B 0,C 180,E1 9695.275,E2 9695.275} C_VEL
LIN {X 0,Y 281.333,Z 642.181,A -85,B 0,C 180,E1 9692.765,E2 9692.765} C_VEL
LIN {X 0,Y 277.831,Z 664.415,A -85,B 0,C 180,E1 9692.094,E2 9692.094} C_VEL
LIN {X 0,Y 273.726,Z 682.317,A -85,B 0,C 180,E1 9691.348,E2 9691.348} C_VEL
LIN {X 0,Y 268.995,Z 699.047,A -85,B 0,C 180,E1 9690.43,E2 9690.43} C_VEL
LIN {X 0,Y 261.86,Z 719.664,A -85,B 0,C 180,E1 9688.941,E2 9688.941} C_VEL
LIN {X 0,Y 255.5,Z 735.171,A -85,B 0,C 180,E1 9687.49,E2 9687.49} C_VEL
LIN {X 0,Y 248.547,Z 750.21,A -85,B 0,C 180,E1 9685.757,E2 9685.757} C_VEL
LIN {X 0,Y 248.141,Z 751.061,A -85,B 0,C 180,E1 9685.65,E2 9685.65} C_VEL
LIN {X 0,Y 244.464,Z 757.33,A -85,B 0,C 180,E1 9685.007,E2 9685.007} C_VEL
LIN {X 0,Y 233.038,Z 771.75,A -85,B 0,C 180,E1 9683.849,E2 9683.849} C_VEL
LIN {X 0,Y 228.8,Z 777.377,A -85,B 0,C 180,E1 9683.038,E2 9683.038} C_VEL
LIN {X 0,Y 228.287,Z 778.147,A -85,B 0,C 180,E1 9682.888,E2 9682.888} C_VEL
LIN {X 0,Y 220.163,Z 790.759,A -85,B 0,C 180,E1 9680.128,E2 9680.128} C_VEL
LIN {X 0,Y 212.081,Z 802.519,A -85,B 0,C 180,E1 9676.947,E2 9676.947} C_VEL
LIN {X 0,Y 203.214,Z 814.79,A -85,B 0,C 180,E1 9672.763,E2 9672.763} C_VEL
LIN {X 0,Y 195.481,Z 824.94,A -85,B 0,C 180,E1 9668.234,E2 9668.234} C_VEL
LIN {X 0,Y 189.345,Z 833.038,A -85,B 0,C 180,E1 9663.673,E2 9663.673} C_VEL
LIN {X 0,Y 183.33,Z 841.341,A -85,B 0,C 180,E1 9657.617,E2 9657.617} C_VEL
LIN {X 0,Y 179.354,Z 847.33,A -85,B 0,C 180,E1 9651.588,E2 9651.588} C_VEL
LIN {X 0,Y 177.185,Z 851.404,A -85,B 0,C 180,E1 9646.051,E2 9646.051} C_VEL
LIN {X 0,Y 176.1,Z 854.708,A -85,B 0,C 180,E1 9639.477,E2 9639.477} C_VEL
LIN {X 0,Y 175.99,Z 856.122,A -85,B 0,C 180,E1 9633.583,E2 9633.583} C_VEL
LIN {X 0,Y 176.02,Z 856.335,A -85,B 0,C 180,E1 9628.698,E2 9628.698} C_VEL
LIN {X 0,Y 175.986,Z 855.529,A -85,B 0,C 180,E1 9623.476,E2 9623.476} C_VEL
LIN {X 0,Y 176.324,Z 853.676,A -85,B 0,C 180,E1 9618.221,E2 9618.221} C_VEL
LIN {X 0,Y 177.584,Z 850.558,A -85,B 0,C 180,E1 9612.639,E2 9612.639} C_VEL
LIN {X 0,Y 180.625,Z 845.381,A -85,B 0,C 180,E1 9606.166,E2 9606.166} C_VEL
LIN {X 0,Y 185.219,Z 838.614,A -85,B 0,C 180,E1 9600.223,E2 9600.223} C_VEL
LIN {X 0,Y 190.408,Z 831.624,A -85,B 0,C 180,E1 9595.451,E2 9595.451} C_VEL
LIN {X 0,Y 197.633,Z 822.216,A -85,B 0,C 180,E1 9590.399,E2 9590.399} C_VEL
LIN {X 0,Y 205.704,Z 811.338,A -85,B 0,C 180,E1 9585.968,E2 9585.968} C_VEL
LIN {X 0,Y 213.191,Z 800.931,A -85,B 0,C 180,E1 9582.583,E2 9582.583} C_VEL
LIN {X 0,Y 221.984,Z 788.082,A -85,B 0,C 180,E1 9579.222,E2 9579.222} C_VEL
LIN {X 0,Y 231.482,Z 772.837,A -85,B 0,C 180,E1 9576.128,E2 9576.128} C_VEL
LIN {X 0,Y 239.206,Z 759.241,A -85,B 0,C 180,E1 9573.934,E2 9573.934} C_VEL
LIN {X 0,Y 246.922,Z 744.276,A -85,B 0,C 180,E1 9571.973,E2 9571.973} C_VEL
LIN {X 0,Y 255.289,Z 725.61,A -85,B 0,C 180,E1 9570.056,E2 9570.056} C_VEL
LIN {X 0,Y 261.29,Z 710.04,A -85,B 0,C 180,E1 9568.804,E2 9568.804} C_VEL
LIN {X 0,Y 266.664,Z 693.831,A -85,B 0,C 180,E1 9567.766,E2 9567.766} C_VEL
LIN {X 0,Y 272.199,Z 673.31,A -85,B 0,C 180,E1 9566.767,E2 9566.767} C_VEL
LIN {X 0,Y 275.94,Z 654.408,A -85,B 0,C 180,E1 9566.11,E2 9566.11} C_VEL
LIN {X 0,Y 278.375,Z 636.339,A -85,B 0,C 180,E1 9565.628,E2 9565.628} C_VEL
LIN {X 0,Y 287.818,Z 528.888,A -85,B 0,C 180,E1 9563.338,E2 9563.338} C_VEL
LIN {X 0,Y 284.007,Z 519.815,A -85,B 0,C 180,E1 9560.89,E2 9560.89} C_VEL
LIN {X 0,Y 279.451,Z 511.643,A -85,B 0,C 180,E1 9557.66,E2 9557.66} C_VEL
LIN {X 0,Y 275.877,Z 505.717,A -85,B 0,C 180,E1 9554.612,E2 9554.612} C_VEL
LIN {X 0,Y 273.596,Z 501.982,A -85,B 0,C 180,E1 9552.246,E2 9552.246} C_VEL
LIN {X 0,Y 271.103,Z 497.817,A -85,B 0,C 180,E1 9548.92,E2 9548.92} C_VEL
LIN {X 0,Y 268.822,Z 493.919,A -85,B 0,C 180,E1 9543.848,E2 9543.848} C_VEL
LIN {X 0,Y 268.545,Z 492.879,A -85,B 0,C 180,E1 9542.356,E2 9542.356} C_VEL
LIN {X 0,Y 268.674,Z 493.045,A -85,B 0,C 180,E1 9536.596,E2 9536.596} C_VEL
LIN {X 0,Y 270.56,Z 497.264,A -85,B 0,C 180,E1 9531.509,E2 9531.509} C_VEL
LIN {X 0,Y 271.519,Z 498.403,A -85,B 0,C 180,E1 9530.043,E2 9530.043} C_VEL
LIN {X 0,Y 274.529,Z 503.512,A -85,B 0,C 180,E1 9526.316,E2 9526.316} C_VEL
LIN {X 0,Y 277.595,Z 508.601,A -85,B 0,C 180,E1 9523.425,E2 9523.425} C_VEL
LIN {X 0,Y 288.536,Z 524.267,A -85,B 0,C 180,E1 9516.201,E2 9516.201} C_VEL
LIN {X 0,Y 298.201,Z 533.33,A -85,B 0,C 180,E1 9511.798,E2 9511.798} C_VEL
LIN {X 0,Y 302.87,Z 536.992,A -85,B 0,C 180,E1 9509.893,E2 9509.893} C_VEL
LIN {X 0,Y 308.474,Z 541.478,A -85,B 0,C 180,E1 9507.461,E2 9507.461} C_VEL
LIN {X 0,Y 312.057,Z 544.321,A -85,B 0,C 180,E1 9505.796,E2 9505.796} C_VEL
LIN {X 0,Y 317.328,Z 548.861,A -85,B 0,C 180,E1 9503.158,E2 9503.158} C_VEL
LIN {X 0,Y 320.88,Z 551.891,A -85,B 0,C 180,E1 9501.167,E2 9501.167} C_VEL
LIN {X 0,Y 326.03,Z 556.833,A -85,B 0,C 180,E1 9498.058,E2 9498.058} C_VEL
LIN {X 0,Y 329.094,Z 559.462,A -85,B 0,C 180,E1 9496.169,E2 9496.169} C_VEL
LIN {X 0,Y 333.919,Z 564.07,A -85,B 0,C 180,E1 9493.078,E2 9493.078} C_VEL
LIN {X 0,Y 337.379,Z 566.84,A -85,B 0,C 180,E1 9490.798,E2 9490.798} C_VEL
LIN {X 0,Y 342.048,Z 571.424,A -85,B 0,C 180,E1 9487.521,E2 9487.521} C_VEL
LIN {X 0,Y 346.239,Z 574.609,A -85,B 0,C 180,E1 9484.471,E2 9484.471} C_VEL
LIN {X 0,Y 349.899,Z 578.366,A -85,B 0,C 180,E1 9481.528,E2 9481.528} C_VEL
LIN {X 0,Y 353.676,Z 581.159,A -85,B 0,C 180,E1 9478.355,E2 9478.355} C_VEL
LIN {X 0,Y 355.396,Z 582.322,A -85,B 0,C 180,E1 9476.825,E2 9476.825} C_VEL
LIN {X 0,Y 358.525,Z 585.797,A -85,B 0,C 180,E1 9473.677,E2 9473.677} C_VEL
LIN {X 0,Y 361.491,Z 588.182,A -85,B 0,C 180,E1 9470.37,E2 9470.37} C_VEL
LIN {X 0,Y 364.235,Z 589.619,A -85,B 0,C 180,E1 9466.916,E2 9466.916} C_VEL
LIN {X 0,Y 365.375,Z 590.404,A -85,B 0,C 180,E1 9465.23,E2 9465.23} C_VEL
LIN {X 0,Y 367.174,Z 592.877,A -85,B 0,C 180,E1 9461.944,E2 9461.944} C_VEL
LIN {X 0,Y 368.532,Z 594.309,A -85,B 0,C 180,E1 9458.739,E2 9458.739} C_VEL
LIN {X 0,Y 369.541,Z 595.212,A -85,B 0,C 180,E1 9455.278,E2 9455.278} C_VEL
LIN {X 0,Y 370.112,Z 595.627,A -85,B 0,C 180,E1 9451.858,E2 9451.858} C_VEL
LIN {X 0,Y 370.106,Z 595.625,A -85,B 0,C 180,E1 9448.607,E2 9448.607} C_VEL
LIN {X 0,Y 369.649,Z 595.289,A -85,B 0,C 180,E1 9445.19,E2 9445.19} C_VEL
LIN {X 0,Y 368.786,Z 594.541,A -85,B 0,C 180,E1 9441.895,E2 9441.895} C_VEL
LIN {X 0,Y 367.458,Z 593.199,A -85,B 0,C 180,E1 9438.702,E2 9438.702} C_VEL
LIN {X 0,Y 365.89,Z 591.125,A -85,B 0,C 180,E1 9435.601,E2 9435.601} C_VEL
LIN {X 0,Y 364.658,Z 589.765,A -85,B 0,C 180,E1 9433.633,E2 9433.633} C_VEL
LIN {X 0,Y 362.067,Z 588.543,A -85,B 0,C 180,E1 9430.304,E2 9430.304} C_VEL
LIN {X 0,Y 359.018,Z 586.274,A -85,B 0,C 180,E1 9426.879,E2 9426.879} C_VEL
LIN {X 0,Y 355.852,Z 582.928,A -85,B 0,C 180,E1 9423.645,E2 9423.645} C_VEL
LIN {X 0,Y 354.622,Z 581.642,A -85,B 0,C 180,E1 9422.459,E2 9422.459} C_VEL
LIN {X 0,Y 350.971,Z 579.256,A -85,B 0,C 180,E1 9419.335,E2 9419.335} C_VEL
LIN {X 0,Y 347.026,Z 575.504,A -85,B 0,C 180,E1 9416.134,E2 9416.134} C_VEL
LIN {X 0,Y 344.928,Z 573.475,A -85,B 0,C 180,E1 9414.524,E2 9414.524} C_VEL
LIN {X 0,Y 340.622,Z 570.148,A -85,B 0,C 180,E1 9411.453,E2 9411.453} C_VEL
LIN {X 0,Y 335.874,Z 565.51,A -85,B 0,C 180,E1 9408.179,E2 9408.179} C_VEL
LIN {X 0,Y 330.944,Z 561.414,A -85,B 0,C 180,E1 9405.013,E2 9405.013} C_VEL
LIN {X 0,Y 327.279,Z 557.771,A -85,B 0,C 180,E1 9402.691,E2 9402.691} C_VEL
LIN {X 0,Y 322.343,Z 553.434,A -85,B 0,C 180,E1 9399.702,E2 9399.702} C_VEL
LIN {X 0,Y 318.872,Z 550.04,A -85,B 0,C 180,E1 9397.681,E2 9397.681} C_VEL
LIN {X 0,Y 313.368,Z 545.527,A -85,B 0,C 180,E1 9394.817,E2 9394.817} C_VEL
LIN {X 0,Y 309.28,Z 542.029,A -85,B 0,C 180,E1 9392.884,E2 9392.884} C_VEL
LIN {X 0,Y 303.472,Z 537.532,A -85,B 0,C 180,E1 9390.369,E2 9390.369} C_VEL
LIN {X 0,Y 298.858,Z 533.794,A -85,B 0,C 180,E1 9388.461,E2 9388.461} C_VEL
LIN {X 0,Y 291.396,Z 527.213,A -85,B 0,C 180,E1 9385.224,E2 9385.224} C_VEL
LIN {X 0,Y 283.961,Z 518.621,A -85,B 0,C 180,E1 9381.199,E2 9381.199} C_VEL
LIN {X 0,Y 276.637,Z 506.83,A -85,B 0,C 180,E1 9375.718,E2 9375.718} C_VEL
LIN {X 0,Y 273.529,Z 501.899,A -85,B 0,C 180,E1 9372.588,E2 9372.588} C_VEL
LIN {X 0,Y 271.102,Z 497.782,A -85,B 0,C 180,E1 9369.329,E2 9369.329} C_VEL
LIN {X 0,Y 268.738,Z 493.488,A -85,B 0,C 180,E1 9363.83,E2 9363.83} C_VEL
LIN {X 0,Y 268.505,Z 492.845,A -85,B 0,C 180,E1 9362.552,E2 9362.552} C_VEL
LIN {X 0,Y 268.67,Z 493.088,A -85,B 0,C 180,E1 9357.004,E2 9357.004} C_VEL
LIN {X 0,Y 270.69,Z 497.433,A -85,B 0,C 180,E1 9351.709,E2 9351.709} C_VEL
LIN {X 0,Y 271.586,Z 498.59,A -85,B 0,C 180,E1 9350.348,E2 9350.348} C_VEL
LIN {X 0,Y 274.637,Z 503.636,A -85,B 0,C 180,E1 9346.625,E2 9346.625} C_VEL
LIN {X 0,Y 277.422,Z 508.334,A -85,B 0,C 180,E1 9343.987,E2 9343.987} C_VEL
LIN {X 0,Y 281.164,Z 514.575,A -85,B 0,C 180,E1 9341.062,E2 9341.062} C_VEL
LIN {X 0,Y 284.738,Z 521.379,A -85,B 0,C 180,E1 9338.627,E2 9338.627} C_VEL
LIN {X 0,Y 287.828,Z 529.129,A -85,B 0,C 180,E1 9336.643,E2 9336.643} C_VEL
LIN {X 0,Y 277.729,Z 642.151,A -85,B 0,C 180,E1 9334.232,E2 9334.232} C_VEL
LIN {X 0,Y 274.042,Z 664.746,A -85,B 0,C 180,E1 9333.556,E2 9333.556} C_VEL
LIN {X 0,Y 269.966,Z 682.08,A -85,B 0,C 180,E1 9332.845,E2 9332.845} C_VEL
LIN {X 0,Y 265.114,Z 698.809,A -85,B 0,C 180,E1 9331.944,E2 9331.944} C_VEL
LIN {X 0,Y 257.814,Z 719.358,A -85,B 0,C 180,E1 9330.484,E2 9330.484} C_VEL
LIN {X 0,Y 251.243,Z 734.932,A -85,B 0,C 180,E1 9329.047,E2 9329.047} C_VEL
LIN {X 0,Y 244.073,Z 749.97,A -85,B 0,C 180,E1 9327.332,E2 9327.332} C_VEL
LIN {X 0,Y 234.799,Z 767.221,A -85,B 0,C 180,E1 9324.843,E2 9324.843} C_VEL
LIN {X 0,Y 228.287,Z 778.147,A -85,B 0,C 180,E1 9322.888,E2 9322.888} C_VEL
LIN {X 0,Y 224.135,Z 783.694,A -85,B 0,C 180,E1 9321.948,E2 9321.948} C_VEL
LIN {X 0,Y 211.128,Z 797.066,A -85,B 0,C 180,E1 9319.94,E2 9319.94} C_VEL
LIN {X 0,Y 206.936,Z 801.778,A -85,B 0,C 180,E1 9318.758,E2 9318.758} C_VEL
LIN {X 0,Y 197.785,Z 813.905,A -85,B 0,C 180,E1 9314.641,E2 9314.641} C_VEL
LIN {X 0,Y 189.091,Z 824.697,A -85,B 0,C 180,E1 9309.776,E2 9309.776} C_VEL
LIN {X 0,Y 182.56,Z 832.795,A -85,B 0,C 180,E1 9305.103,E2 9305.103} C_VEL
LIN {X 0,Y 176.095,Z 841.098,A -85,B 0,C 180,E1 9298.856,E2 9298.856} C_VEL
LIN {X 0,Y 171.768,Z 847.089,A -85,B 0,C 180,E1 9292.592,E2 9292.592} C_VEL
LIN {X 0,Y 169.369,Z 851.163,A -85,B 0,C 180,E1 9286.814,E2 9286.814} C_VEL
LIN {X 0,Y 168.131,Z 854.469,A -85,B 0,C 180,E1 9279.931,E2 9279.931} C_VEL
LIN {X 0,Y 167.99,Z 855.886,A -85,B 0,C 180,E1 9273.754,E2 9273.754} C_VEL
LIN {X 0,Y 168.022,Z 856.099,A -85,B 0,C 180,E1 9268.636,E2 9268.636} C_VEL
LIN {X 0,Y 167.987,Z 855.381,A -85,B 0,C 180,E1 9263.507,E2 9263.507} C_VEL
LIN {X 0,Y 168.345,Z 853.588,A -85,B 0,C 180,E1 9258.002,E2 9258.002} C_VEL
LIN {X 0,Y 169.696,Z 850.529,A -85,B 0,C 180,E1 9252.159,E2 9252.159} C_VEL
LIN {X 0,Y 172.946,Z 845.447,A -85,B 0,C 180,E1 9245.402,E2 9245.402} C_VEL
LIN {X 0,Y 177.828,Z 838.773,A -85,B 0,C 180,E1 9239.227,E2 9239.227} C_VEL
LIN {X 0,Y 183.312,Z 831.852,A -85,B 0,C 180,E1 9234.296,E2 9234.296} C_VEL
LIN {X 0,Y 190.446,Z 823.064,A -85,B 0,C 180,E1 9229.384,E2 9229.384} C_VEL
LIN {X 0,Y 199.354,Z 811.799,A -85,B 0,C 180,E1 9224.588,E2 9224.588} C_VEL
LIN {X 0,Y 207.152,Z 801.483,A -85,B 0,C 180,E1 9221.154,E2 9221.154} C_VEL
LIN {X 0,Y 215.641,Z 789.625,A -85,B 0,C 180,E1 9217.981,E2 9217.981} C_VEL
LIN {X 0,Y 226.098,Z 773.719,A -85,B 0,C 180,E1 9214.663,E2 9214.663} C_VEL
LIN {X 0,Y 234.412,Z 759.632,A -85,B 0,C 180,E1 9212.379,E2 9212.379} C_VEL
LIN {X 0,Y 241.99,Z 745.46,A -85,B 0,C 180,E1 9210.519,E2 9210.519} C_VEL
LIN {X 0,Y 250.626,Z 727.106,A -85,B 0,C 180,E1 9208.612,E2 9208.612} C_VEL
LIN {X 0,Y 257.074,Z 710.971,A -85,B 0,C 180,E1 9207.315,E2 9207.315} C_VEL
LIN {X 0,Y 262.613,Z 694.838,A -85,B 0,C 180,E1 9206.285,E2 9206.285} C_VEL
LIN {X 0,Y 268.017,Z 675.895,A -85,B 0,C 180,E1 9205.351,E2 9205.351} C_VEL
LIN {X 0,Y 272.32,Z 655.257,A -85,B 0,C 180,E1 9204.626,E2 9204.626} C_VEL
LIN {X 0,Y 274.832,Z 637.54,A -85,B 0,C 180,E1 9204.154,E2 9204.154} C_VEL
LIN {X 0,Y 284.313,Z 532.85,A -85,B 0,C 180,E1 9201.922,E2 9201.922} C_VEL
LIN {X 0,Y 281.378,Z 525.852,A -85,B 0,C 180,E1 9199.9,E2 9199.9} C_VEL
LIN {X 0,Y 277.133,Z 518.036,A -85,B 0,C 180,E1 9196.676,E2 9196.676} C_VEL
LIN {X 0,Y 273.926,Z 512.581,A -85,B 0,C 180,E1 9193.733,E2 9193.733} C_VEL
LIN {X 0,Y 272.158,Z 509.553,A -85,B 0,C 180,E1 9191.773,E2 9191.773} C_VEL
LIN {X 0,Y 269.99,Z 505.695,A -85,B 0,C 180,E1 9188.742,E2 9188.742} C_VEL
LIN {X 0,Y 267.785,Z 501.816,A -85,B 0,C 180,E1 9183.648,E2 9183.648} C_VEL
LIN {X 0,Y 267.57,Z 500.827,A -85,B 0,C 180,E1 9182.365,E2 9182.365} C_VEL
LIN {X 0,Y 267.649,Z 500.962,A -85,B 0,C 180,E1 9176.797,E2 9176.797} C_VEL
LIN {X 0,Y 269.587,Z 505.277,A -85,B 0,C 180,E1 9171.478,E2 9171.478} C_VEL
LIN {X 0,Y 270.381,Z 506.419,A -85,B 0,C 180,E1 9170.216,E2 9170.216} C_VEL
LIN {X 0,Y 273.054,Z 511.062,A -85,B 0,C 180,E1 9166.78,E2 9166.78} C_VEL
LIN {X 0,Y 275.952,Z 516.067,A -85,B 0,C 180,E1 9163.918,E2 9163.918} C_VEL
LIN {X 0,Y 286.518,Z 531.635,A -85,B 0,C 180,E1 9156.678,E2 9156.678} C_VEL
LIN {X 0,Y 296.217,Z 540.874,A -85,B 0,C 180,E1 9152.14,E2 9152.14} C_VEL
LIN {X 0,Y 301.362,Z 544.92,A -85,B 0,C 180,E1 9150.056,E2 9150.056} C_VEL
LIN {X 0,Y 307.401,Z 549.609,A -85,B 0,C 180,E1 9147.444,E2 9147.444} C_VEL
LIN {X 0,Y 310.807,Z 552.435,A -85,B 0,C 180,E1 9145.863,E2 9145.863} C_VEL
LIN {X 0,Y 316.187,Z 556.897,A -85,B 0,C 180,E1 9143.197,E2 9143.197} C_VEL
LIN {X 0,Y 319.46,Z 559.729,A -85,B 0,C 180,E1 9141.375,E2 9141.375} C_VEL
LIN {X 0,Y 324.591,Z 564.577,A -85,B 0,C 180,E1 9138.304,E2 9138.304} C_VEL
LIN {X 0,Y 327.664,Z 567.225,A -85,B 0,C 180,E1 9136.413,E2 9136.413} C_VEL
LIN {X 0,Y 332.601,Z 571.887,A -85,B 0,C 180,E1 9133.266,E2 9133.266} C_VEL
LIN {X 0,Y 336.131,Z 574.755,A -85,B 0,C 180,E1 9130.943,E2 9130.943} C_VEL
LIN {X 0,Y 340.931,Z 579.379,A -85,B 0,C 180,E1 9127.589,E2 9127.589} C_VEL
LIN {X 0,Y 345.008,Z 582.492,A -85,B 0,C 180,E1 9124.627,E2 9124.627} C_VEL
LIN {X 0,Y 348.891,Z 586.387,A -85,B 0,C 180,E1 9121.527,E2 9121.527} C_VEL
LIN {X 0,Y 352.573,Z 589.06,A -85,B 0,C 180,E1 9118.452,E2 9118.452} C_VEL
LIN {X 0,Y 354.295,Z 590.268,A -85,B 0,C 180,E1 9116.925,E2 9116.925} C_VEL
LIN {X 0,Y 357.449,Z 593.725,A -85,B 0,C 180,E1 9113.752,E2 9113.752} C_VEL
LIN {X 0,Y 360.478,Z 596.128,A -85,B 0,C 180,E1 9110.393,E2 9110.393} C_VEL
LIN {X 0,Y 363.213,Z 597.548,A -85,B 0,C 180,E1 9106.965,E2 9106.965} C_VEL
LIN {X 0,Y 364.362,Z 598.366,A -85,B 0,C 180,E1 9105.274,E2 9105.274} C_VEL
LIN {X 0,Y 366.104,Z 600.733,A -85,B 0,C 180,E1 9102.139,E2 9102.139} C_VEL
LIN {X 0,Y 367.473,Z 602.202,A -85,B 0,C 180,E1 9098.922,E2 9098.922} C_VEL
LIN {X 0,Y 368.533,Z 603.129,A -85,B 0,C 180,E1 9095.433,E2 9095.433} C_VEL
LIN {X 0,Y 369.12,Z 603.555,A -85,B 0,C 180,E1 9092.018,E2 9092.018} C_VEL
LIN {X 0,Y 369.133,Z 603.558,A -85,B 0,C 180,E1 9088.758,E2 9088.758} C_VEL
LIN {X 0,Y 368.71,Z 603.253,A -85,B 0,C 180,E1 9085.334,E2 9085.334} C_VEL
LIN {X 0,Y 367.846,Z 602.538,A -85,B 0,C 180,E1 9082.032,E2 9082.032} C_VEL
LIN {X 0,Y 366.534,Z 601.231,A -85,B 0,C 180,E1 9078.833,E2 9078.833} C_VEL
LIN {X 0,Y 364.984,Z 599.229,A -85,B 0,C 180,E1 9075.727,E2 9075.727} C_VEL
LIN {X 0,Y 363.659,Z 597.701,A -85,B 0,C 180,E1 9073.61,E2 9073.61} C_VEL
LIN {X 0,Y 361.04,Z 596.472,A -85,B 0,C 180,E1 9070.254,E2 9070.254} C_VEL
LIN {X 0,Y 358.125,Z 594.351,A -85,B 0,C 180,E1 9066.992,E2 9066.992} C_VEL
LIN {X 0,Y 354.955,Z 591.117,A -85,B 0,C 180,E1 9063.754,E2 9063.754} C_VEL
LIN {X 0,Y 353.425,Z 589.501,A -85,B 0,C 180,E1 9062.289,E2 9062.289} C_VEL
LIN {X 0,Y 349.833,Z 587.158,A -85,B 0,C 180,E1 9059.231,E2 9059.231} C_VEL
LIN {X 0,Y 345.882,Z 583.469,A -85,B 0,C 180,E1 9056.043,E2 9056.043} C_VEL
LIN {X 0,Y 343.782,Z 581.378,A -85,B 0,C 180,E1 9054.432,E2 9054.432} C_VEL
LIN {X 0,Y 339.392,Z 578.025,A -85,B 0,C 180,E1 9051.308,E2 9051.308} C_VEL
LIN {X 0,Y 334.513,Z 573.299,A -85,B 0,C 180,E1 9047.97,E2 9047.97} C_VEL
LIN {X 0,Y 329.519,Z 569.158,A -85,B 0,C 180,E1 9044.765,E2 9044.765} C_VEL
LIN {X 0,Y 325.684,Z 565.406,A -85,B 0,C 180,E1 9042.352,E2 9042.352} C_VEL
LIN {X 0,Y 320.575,Z 560.876,A -85,B 0,C 180,E1 9039.269,E2 9039.269} C_VEL
LIN {X 0,Y 317.017,Z 557.532,A -85,B 0,C 180,E1 9037.256,E2 9037.256} C_VEL
LIN {X 0,Y 311.357,Z 552.945,A -85,B 0,C 180,E1 9034.403,E2 9034.403} C_VEL
LIN {X 0,Y 307.599,Z 549.743,A -85,B 0,C 180,E1 9032.643,E2 9032.643} C_VEL
LIN {X 0,Y 301.761,Z 545.274,A -85,B 0,C 180,E1 9030.119,E2 9030.119} C_VEL
LIN {X 0,Y 296.649,Z 541.185,A -85,B 0,C 180,E1 9028.035,E2 9028.035} C_VEL
LIN {X 0,Y 289.135,Z 534.366,A -85,B 0,C 180,E1 9024.67,E2 9024.67} C_VEL
LIN {X 0,Y 282.053,Z 525.995,A -85,B 0,C 180,E1 9020.697,E2 9020.697} C_VEL
LIN {X 0,Y 274.973,Z 514.229,A -85,B 0,C 180,E1 9015.167,E2 9015.167} C_VEL
LIN {X 0,Y 272.154,Z 509.55,A -85,B 0,C 180,E1 9012.185,E2 9012.185} C_VEL
LIN {X 0,Y 269.99,Z 505.66,A -85,B 0,C 180,E1 9009.153,E2 9009.153} C_VEL
LIN {X 0,Y 267.708,Z 501.398,A -85,B 0,C 180,E1 9003.631,E2 9003.631} C_VEL
LIN {X 0,Y 267.494,Z 500.768,A -85,B 0,C 180,E1 9002.347,E2 9002.347} C_VEL
LIN {X 0,Y 267.646,Z 500.999,A -85,B 0,C 180,E1 8997.207,E2 8997.207} C_VEL
LIN {X 0,Y 269.586,Z 505.311,A -85,B 0,C 180,E1 8991.889,E2 8991.889} C_VEL
LIN {X 0,Y 270.382,Z 506.444,A -85,B 0,C 180,E1 8990.627,E2 8990.627} C_VEL
LIN {X 0,Y 273.157,Z 511.183,A -85,B 0,C 180,E1 8987.09,E2 8987.09} C_VEL
LIN {X 0,Y 275.895,Z 516.003,A -85,B 0,C 180,E1 8984.382,E2 8984.382} C_VEL
LIN {X 0,Y 279.337,Z 522.003,A -85,B 0,C 180,E1 8981.578,E2 8981.578} C_VEL
LIN {X 0,Y 282.569,Z 528.44,A -85,B 0,C 180,E1 8979.269,E2 8979.269} C_VEL
LIN {X 0,Y 284.349,Z 533.172,A -85,B 0,C 180,E1 8978.039,E2 8978.039} C_VEL
LIN {X 0,Y 274.336,Z 641.924,A -85,B 0,C 180,E1 8975.742,E2 8975.742} C_VEL
LIN {X 0,Y 270.537,Z 664.63,A -85,B 0,C 180,E1 8975.074,E2 8975.074} C_VEL
LIN {X 0,Y 266.395,Z 681.842,A -85,B 0,C 180,E1 8974.383,E2 8974.383} C_VEL
LIN {X 0,Y 261.424,Z 698.571,A -85,B 0,C 180,E1 8973.501,E2 8973.501} C_VEL
LIN {X 0,Y 253.977,Z 719.014,A -85,B 0,C 180,E1 8972.079,E2 8972.079} C_VEL
LIN {X 0,Y 247.179,Z 734.692,A -85,B 0,C 180,E1 8970.656,E2 8970.656} C_VEL
LIN {X 0,Y 239.792,Z 749.73,A -85,B 0,C 180,E1 8968.964,E2 8968.964} C_VEL
LIN {X 0,Y 230.208,Z 766.98,A -85,B 0,C 180,E1 8966.5,E2 8966.5} C_VEL
LIN {X 0,Y 221.421,Z 780.988,A -85,B 0,C 180,E1 8963.928,E2 8963.928} C_VEL
LIN {X 0,Y 213.153,Z 793.194,A -85,B 0,C 180,E1 8961.137,E2 8961.137} C_VEL
LIN {X 0,Y 206.936,Z 801.778,A -85,B 0,C 180,E1 8958.758,E2 8958.758} C_VEL
LIN {X 0,Y 202.732,Z 806.519,A -85,B 0,C 180,E1 8957.484,E2 8957.484} C_VEL
LIN {X 0,Y 189.445,Z 817.624,A -85,B 0,C 180,E1 8954.497,E2 8954.497} C_VEL
LIN {X 0,Y 185.36,Z 821.62,A -85,B 0,C 180,E1 8952.894,E2 8952.894} C_VEL
LIN {X 0,Y 177.111,Z 831.138,A -85,B 0,C 180,E1 8947.566,E2 8947.566} C_VEL
LIN {X 0,Y 171.15,Z 838.128,A -85,B 0,C 180,E1 8942.51,E2 8942.51} C_VEL
LIN {X 0,Y 165.57,Z 845.151,A -85,B 0,C 180,E1 8935.843,E2 8935.843} C_VEL
LIN {X 0,Y 162.081,Z 850.076,A -85,B 0,C 180,E1 8929.083,E2 8929.083} C_VEL
LIN {X 0,Y 160.476,Z 853.197,A -85,B 0,C 180,E1 8922.961,E2 8922.961} C_VEL
LIN {X 0,Y 160.006,Z 855.053,A -85,B 0,C 180,E1 8917.179,E2 8917.179} C_VEL
LIN {X 0,Y 160.019,Z 855.832,A -85,B 0,C 180,E1 8911.79,E2 8911.79} C_VEL
LIN {X 0,Y 159.999,Z 855.711,A -85,B 0,C 180,E1 8906.776,E2 8906.776} C_VEL
LIN {X 0,Y 160.049,Z 854.69,A -85,B 0,C 180,E1 8901.377,E2 8901.377} C_VEL
LIN {X 0,Y 161.037,Z 852.035,A -85,B 0,C 180,E1 8894.276,E2 8894.276} C_VEL
LIN {X 0,Y 163.705,Z 847.607,A -85,B 0,C 180,E1 8887.288,E2 8887.288} C_VEL
LIN {X 0,Y 167.526,Z 842.54,A -85,B 0,C 180,E1 8881.481,E2 8881.481} C_VEL
LIN {X 0,Y 173.608,Z 835.309,A -85,B 0,C 180,E1 8875.239,E2 8875.239} C_VEL
LIN {X 0,Y 181.459,Z 826.087,A -85,B 0,C 180,E1 8869.445,E2 8869.445} C_VEL
LIN {X 0,Y 188.88,Z 817.334,A -85,B 0,C 180,E1 8865.196,E2 8865.196} C_VEL
LIN {X 0,Y 197.685,Z 806.629,A -85,B 0,C 180,E1 8861.097,E2 8861.097} C_VEL
LIN {X 0,Y 208.118,Z 792.952,A -85,B 0,C 180,E1 8857.109,E2 8857.109} C_VEL
LIN {X 0,Y 216.717,Z 780.747,A -85,B 0,C 180,E1 8854.328,E2 8854.328} C_VEL
LIN {X 0,Y 225.819,Z 766.74,A -85,B 0,C 180,E1 8851.778,E2 8851.778} C_VEL
LIN {X 0,Y 235.714,Z 749.491,A -85,B 0,C 180,E1 8849.347,E2 8849.347} C_VEL
LIN {X 0,Y 243.385,Z 734.31,A -85,B 0,C 180,E1 8847.669,E2 8847.669} C_VEL
LIN {X 0,Y 251.135,Z 716.842,A -85,B 0,C 180,E1 8846.134,E2 8846.134} C_VEL
LIN {X 0,Y 258.204,Z 697.501,A -85,B 0,C 180,E1 8844.852,E2 8844.852} C_VEL
LIN {X 0,Y 263.041,Z 681.531,A -85,B 0,C 180,E1 8844.036,E2 8844.036} C_VEL
LIN {X 0,Y 267.542,Z 663.123,A -85,B 0,C 180,E1 8843.322,E2 8843.322} C_VEL
LIN {X 0,Y 271.16,Z 641.413,A -85,B 0,C 180,E1 8842.706,E2 8842.706} C_VEL
LIN {X 0,Y 281.036,Z 537.142,A -85,B 0,C 180,E1 8840.522,E2 8840.522} C_VEL
